KUKA KRL program: MyProgram_284().src

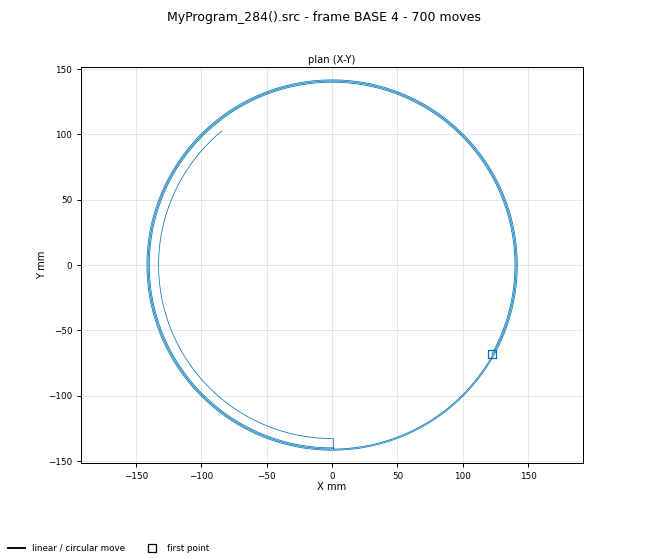
[picture p0: tool path of MyProgram_284().src in frame BASE 4, 700 of 700 moves have a stored position in this frame; points joined in program order, loops and branches not executed]
&ACCESS RVP
&REL 1
&PARAM TEMPLATE = C:\KRC\Roboter\Template\vorgabe
&PARAM EDITMASK = *
DEF MyProgram_284()
; ---- Setting reference (Base) ----
$BASE = BASE_DATA[4]

; --------------------------
; ---- Setting tool (TCP) ----
$TOOL = TOOL_DATA[3]
; --------------------------

$VEL.CP = VEL_APROX_PRINT
Startdeposition()
$VEL.CP = VEL_PRINT
LIN {X 122.1993,Y -68.1495,Z 174,A -26.2551,B 7.7078,C 0.3215,E1 7.8551,E2 478.0769} C_DIS
LIN {X 124.5651,Y -63.7171,Z 174,A -24.1572,B 7.7081,C 0.3154,E1 7.8578,E2 475.9716} C_DIS
LIN {X 126.1549,Y -60.5084,Z 174,A -22.4865,B 7.7084,C 0.3073,E1 7.8599,E2 474.2724} C_DIS
LIN {X 127.9066,Y -56.7133,Z 174,A -21.1789,B 7.7083,C 0.311,E1 7.8613,E2 473.0165} C_DIS
LIN {X 129.634,Y -52.6447,Z 174,A -19.4311,B 7.7083,C 0.3074,E1 7.8632,E2 471.2751} C_DIS
LIN {X 131.5394,Y -47.684,Z 174,A -17.3231,B 7.7086,C 0.3029,E1 7.8652,E2 469.1739} C_DIS
LIN {X 132.6761,Y -44.4231,Z 174,A -15.9508,B 7.7086,C 0.2999,E1 7.8665,E2 467.8057} C_DIS
LIN {X 133.516,Y -41.8378,Z 174,A -14.7782,B 7.7089,C 0.2956,E1 7.8675,E2 466.6243} C_DIS
LIN {X 135.2272,Y -35.9162,Z 174,A -12.5229,B 7.7089,C 0.294,E1 7.8692,E2 464.4017} C_DIS
LIN {X 136.3459,Y -31.4041,Z 174,A -10.4646,B 7.7092,C 0.2855,E1 7.8705,E2 462.3215} C_DIS
LIN {X 137.1536,Y -27.6644,Z 174,A -8.7503,B 7.7095,C 0.278,E1 7.8715,E2 460.5863} C_DIS
LIN {X 138.1088,Y -22.4214,Z 174,A -6.7596,B 7.7095,C 0.2757,E1 7.8725,E2 458.6188} C_DIS
LIN {X 138.6815,Y -18.5466,Z 174,A -5.2004,B 7.7097,C 0.2721,E1 7.8731,E2 457.0639} C_DIS
LIN {X 139.1996,Y -14.1607,Z 174,A -3.1875,B 7.71,C 0.2626,E1 7.8737,E2 455.0226} C_DIS
LIN {X 139.4882,Y -10.9545,Z 174,A -1.9592,B 7.7101,C 0.2607,E1 7.8739,E2 453.8049} C_DIS
LIN {X 139.7863,Y -6.0486,Z 174,A -0.0924,B 7.7102,C 0.2579,E1 7.8742,E2 451.9554} C_DIS
LIN {X 139.9098,Y -1.4915,Z 174,A 1.6918,B 7.7103,C 0.2542,E1 7.8742,E2 450.1803} C_DIS
LIN {X 139.8656,Y 3.7505,Z 174,A 3.9953,B 7.7106,C 0.2448,E1 7.8742,E2 447.8544} C_DIS
LIN {X 139.6455,Y 8.6938,Z 174,A 5.8419,B 7.7106,C 0.2427,E1 7.8739,E2 446.0296} C_DIS
LIN {X 139.3207,Y 12.8988,Z 174,A 7.2965,B 7.7106,C 0.2433,E1 7.8736,E2 444.6089} C_DIS
LIN {X 138.8413,Y 17.3162,Z 174,A 9.4268,B 7.711,C 0.2317,E1 7.8729,E2 442.4369} C_DIS
LIN {X 137.6741,Y 24.9464,Z 174,A 12.3433,B 7.7111,C 0.2278,E1 7.8716,E2 439.5497} C_DIS
LIN {X 136.0253,Y 32.7637,Z 174,A 15.5132,B 7.7113,C 0.2207,E1 7.8697,E2 436.3907} C_DIS
LIN {X 135.2183,Y 35.9496,Z 174,A 16.8457,B 7.7114,C 0.2172,E1 7.8688,E2 435.0589} C_DIS
LIN {X 134.3574,Y 39.045,Z 174,A 18.167,B 7.7116,C 0.2135,E1 7.8678,E2 433.7359} C_DIS
LIN {X 133.4759,Y 41.9634,Z 174,A 19.4631,B 7.7116,C 0.2091,E1 7.8667,E2 432.4328} C_DIS
LIN {X 132.2647,Y 45.6334,Z 174,A 20.9077,B 7.7117,C 0.2076,E1 7.8654,E2 431.0049} C_DIS
LIN {X 131.2197,Y 48.5594,Z 174,A 22.2206,B 7.7118,C 0.2033,E1 7.8641,E2 429.686} C_DIS
LIN {X 129.941,Y 51.8831,Z 174,A 24.4494,B 7.7123,C 0.1838,E1 7.8617,E2 427.3561} C_DIS
LIN {X 127.4014,Y 57.8428,Z 174,A 26.6346,B 7.7123,C 0.1864,E1 7.8593,E2 425.2304} C_DIS
LIN {X 125.7153,Y 61.4186,Z 174,A 27.8606,B 7.7122,C 0.1901,E1 7.8579,E2 424.0542} C_DIS
LIN {X 124.1071,Y 64.6062,Z 174,A 29.3051,B 7.7122,C 0.1868,E1 7.856,E2 422.6111} C_DIS
LIN {X 122.3418,Y 67.8921,Z 174,A 31.3586,B 7.7126,C 0.1724,E1 7.8531,E2 420.4888} C_DIS
LIN {X 119.7806,Y 72.315,Z 174,A 32.9061,B 7.7124,C 0.1782,E1 7.851,E2 419.0109} C_DIS
LIN {X 117.2705,Y 76.3185,Z 174,A 34.6702,B 7.7124,C 0.1769,E1 7.8484,E2 417.2678} C_DIS
LIN {X 115.0409,Y 79.6401,Z 174,A 36.4617,B 7.7126,C 0.17,E1 7.8456,E2 415.4559} C_DIS
LIN {X 112.3183,Y 83.4354,Z 174,A 38.1328,B 7.7126,C 0.1703,E1 7.8429,E2 413.8149} C_DIS
LIN {X 110.0921,Y 86.3509,Z 174,A 40.1246,B 7.7129,C 0.1573,E1 7.8393,E2 411.7595} C_DIS
LIN {X 107.4607,Y 89.6059,Z 174,A 41.515,B 7.7129,C 0.1599,E1 7.8369,E2 410.4102} C_DIS
LIN {X 104.7041,Y 92.8113,Z 174,A 43.4594,B 7.713,C 0.152,E1 7.8333,E2 408.4378} C_DIS
LIN {X 102.1452,Y 95.6208,Z 174,A 44.6972,B 7.713,C 0.1549,E1 7.831,E2 407.2404} C_DIS
LIN {X 99.0411,Y 98.8322,Z 174,A 46.4208,B 7.713,C 0.1532,E1 7.8277,E2 405.5298} C_DIS
LIN {X 94.8635,Y 102.8485,Z 174,A 48.8946,B 7.7131,C 0.1466,E1 7.8226,E2 403.0426} C_DIS
LIN {X 91.3702,Y 105.9639,Z 174,A 50.7297,B 7.7131,C 0.1446,E1 7.8188,E2 401.2174} C_DIS
LIN {X 88.0563,Y 108.7337,Z 174,A 52.5226,B 7.7132,C 0.1409,E1 7.8149,E2 399.421} C_DIS
LIN {X 84.604,Y 111.4413,Z 174,A 54.3131,B 7.7132,C 0.1379,E1 7.8109,E2 397.6311} C_DIS
LIN {X 80.4569,Y 114.4709,Z 174,A 56.6668,B 7.7134,C 0.1296,E1 7.8055,E2 395.2449} C_DIS
LIN {X 77.2065,Y 116.6881,Z 174,A 57.992,B 7.7134,C 0.1325,E1 7.8025,E2 393.9562} C_DIS
LIN {X 73.4825,Y 119.0685,Z 174,A 59.8229,B 7.7134,C 0.1293,E1 7.7982,E2 392.1225} C_DIS
LIN {X 69.1583,Y 121.6306,Z 174,A 61.7597,B 7.7134,C 0.1286,E1 7.7935,E2 390.2011} C_DIS
LIN {X 66.0546,Y 123.3437,Z 174,A 63.2273,B 7.7134,C 0.1264,E1 7.7899,E2 388.7314} C_DIS
LIN {X 58.451,Y 127.1215,Z 174,A 66.6086,B 7.7135,C 0.1238,E1 7.7815,E2 385.3624} C_DIS
LIN {X 52.7496,Y 129.5917,Z 174,A 69.091,B 7.7135,C 0.1221,E1 7.7751,E2 382.8883} C_DIS
LIN {X 49.4162,Y 130.8987,Z 174,A 70.6147,B 7.7135,C 0.1195,E1 7.7711,E2 381.3573} C_DIS
LIN {X 46.0839,Y 132.1085,Z 174,A 71.9894,B 7.7135,C 0.1195,E1 7.7675,E2 379.9926} C_DIS
LIN {X 43.2163,Y 133.0757,Z 174,A 73.315,B 7.7136,C 0.1169,E1 7.764,E2 378.6564} C_DIS
LIN {X 39.8202,Y 134.1304,Z 174,A 74.7349,B 7.7136,C 0.1163,E1 7.7602,E2 377.2413} C_DIS
LIN {X 36.1319,Y 135.1697,Z 174,A 76.2357,B 7.7136,C 0.1163,E1 7.7562,E2 375.7495} C_DIS
LIN {X 32.151,Y 136.1728,Z 174,A 78.6804,B 7.7138,C 0.1016,E1 7.7493,E2 373.2079} C_DIS
LIN {X 26.4354,Y 137.3957,Z 174,A 80.31,B 7.7137,C 0.1138,E1 7.7451,E2 371.6764} C_DIS
LIN {X 19.3821,Y 138.5673,Z 174,A 83.3147,B 7.7137,C 0.1112,E1 7.7368,E2 368.663} C_DIS
LIN {X 13.9273,Y 139.222,Z 174,A 85.559,B 7.7137,C 0.1106,E1 7.7306,E2 366.4202} C_DIS
LIN {X 10.1279,Y 139.5487,Z 174,A 87.0357,B 7.7137,C 0.1117,E1 7.7265,E2 364.9547} C_DIS
LIN {X 5.4892,Y 139.8081,Z 174,A 89.1817,B 7.7137,C 0.1073,E1 7.7204,E2 362.7787} C_DIS
LIN {X 0.3109,Y 139.9163,Z 174,A 91.1091,B 7.7137,C 0.1105,E1 7.7151,E2 360.8768} C_DIS
LIN {X -3.9902,Y 139.859,Z 174,A 92.7867,B 7.7137,C 0.112,E1 7.7104,E2 359.2106} C_DIS
LIN {X -9.1606,Y 139.6167,Z 174,A 94.922,B 7.7137,C 0.1121,E1 7.7045,E2 357.0744} C_DIS
LIN {X -14.8422,Y 139.1263,Z 174,A 97.3717,B 7.7137,C 0.1108,E1 7.6976,E2 354.6115} C_DIS
LIN {X -19.4903,Y 138.5519,Z 174,A 99.8517,B 7.7138,C 0.1022,E1 7.6906,E2 352.0612} C_DIS
LIN {X -24.6926,Y 137.7195,Z 174,A 101.2095,B 7.7136,C 0.1165,E1 7.6871,E2 350.8061} C_DIS
LIN {X -27.3108,Y 137.2255,Z 174,A 102.6319,B 7.7136,C 0.1117,E1 7.6831,E2 349.3427} C_DIS
LIN {X -32.0121,Y 136.2065,Z 174,A 104.56,B 7.7136,C 0.1136,E1 7.6779,E2 347.4211} C_DIS
LIN {X -35.8048,Y 135.2569,Z 174,A 106.0409,B 7.7136,C 0.1167,E1 7.6739,E2 345.9564} C_DIS
LIN {X -39.1445,Y 134.3282,Z 174,A 107.4312,B 7.7136,C 0.1183,E1 7.6702,E2 344.5707} C_DIS
LIN {X -42.3981,Y 133.337,Z 174,A 108.8728,B 7.7136,C 0.1187,E1 7.6663,E2 343.1239} C_DIS
LIN {X -45.0988,Y 132.4501,Z 174,A 110.163,B 7.7136,C 0.1178,E1 7.6629,E2 341.8187} C_DIS
LIN {X -50.4383,Y 130.5081,Z 174,A 113.0061,B 7.7136,C 0.1119,E1 7.6553,E2 338.9116} C_DIS
LIN {X -55.163,Y 128.5827,Z 174,A 114.3244,B 7.7135,C 0.1265,E1 7.6522,E2 337.6926} C_DIS
LIN {X -61.6152,Y 125.6183,Z 174,A 117.4422,B 7.7135,C 0.1268,E1 7.6442,E2 334.5507} C_DIS
LIN {X -64.8167,Y 123.9965,Z 174,A 118.9194,B 7.7135,C 0.1286,E1 7.6405,E2 333.0738} C_DIS
LIN {X -67.5389,Y 122.5374,Z 174,A 120.7434,B 7.7135,C 0.1217,E1 7.6359,E2 331.18} C_DIS
LIN {X -71.6524,Y 120.1781,Z 174,A 122.2439,B 7.7134,C 0.1314,E1 7.6324,E2 329.7372} C_DIS
LIN {X -74.8429,Y 118.2177,Z 174,A 123.8797,B 7.7134,C 0.1322,E1 7.6285,E2 328.0898} C_DIS
LIN {X -79.0031,Y 115.479,Z 174,A 125.8589,B 7.7133,C 0.1364,E1 7.624,E2 326.12} C_DIS
LIN {X -81.9231,Y 113.4262,Z 174,A 127.1872,B 7.7133,C 0.1409,E1 7.621,E2 324.8098} C_DIS
LIN {X -85.236,Y 110.9577,Z 174,A 129.4591,B 7.7133,C 0.1351,E1 7.6158,E2 322.4658} C_DIS
LIN {X -88.7884,Y 108.1368,Z 174,A 130.9257,B 7.7131,C 0.1444,E1 7.6127,E2 321.0506} C_DIS
LIN {X -94.8734,Y 102.8394,Z 174,A 134.9758,B 7.7132,C 0.1396,E1 7.6041,E2 316.9084} C_DIS
LIN {X -99.2376,Y 98.6344,Z 174,A 136.7497,B 7.7129,C 0.1553,E1 7.6008,E2 315.2271} C_DIS
LIN {X -104.5185,Y 93.021,Z 174,A 140.4374,B 7.7129,C 0.1541,E1 7.5937,E2 311.4749} C_DIS
LIN {X -107.56,Y 89.4863,Z 174,A 141.9414,B 7.7127,C 0.1644,E1 7.5911,E2 310.0243} C_DIS
LIN {X -110.7442,Y 85.5136,Z 174,A 144.0936,B 7.7127,C 0.1681,E1 7.5874,E2 307.8657} C_DIS
LIN {X -113.4608,Y 81.8753,Z 174,A 145.8871,B 7.7126,C 0.1734,E1 7.5844,E2 306.0823} C_DIS
LIN {X -115.9587,Y 78.2972,Z 174,A 147.7171,B 7.7125,C 0.1771,E1 7.5815,E2 304.2486} C_DIS
LIN {X -119.4121,Y 72.9224,Z 174,A 150.4658,B 7.7124,C 0.1816,E1 7.5774,E2 301.4856} C_DIS
LIN {X -121.5604,Y 69.2814,Z 174,A 152.2284,B 7.7123,C 0.1855,E1 7.5749,E2 299.7208} C_DIS
LIN {X -123.7428,Y 65.2999,Z 174,A 153.9528,B 7.7121,C 0.1921,E1 7.5727,E2 298.0153} C_DIS
LIN {X -125.3067,Y 62.2467,Z 174,A 155.2919,B 7.712,C 0.1967,E1 7.571,E2 296.6858} C_DIS
LIN {X -127.1646,Y 58.3576,Z 174,A 157.2294,B 7.712,C 0.1989,E1 7.5687,E2 294.7282} C_DIS
LIN {X -128.8679,Y 54.4954,Z 174,A 159.0105,B 7.7118,C 0.2027,E1 7.5667,E2 292.9421} C_DIS
LIN {X -130.2987,Y 50.9768,Z 174,A 160.5654,B 7.7118,C 0.2069,E1 7.5651,E2 291.3888} C_DIS
LIN {X -131.5535,Y 47.645,Z 174,A 161.9957,B 7.7116,C 0.2113,E1 7.5637,E2 289.9634} C_DIS
LIN {X -132.5578,Y 44.7784,Z 174,A 163.4094,B 7.7116,C 0.2123,E1 7.5624,E2 288.5293} C_DIS
LIN {X -133.7726,Y 41.0028,Z 174,A 164.8584,B 7.7114,C 0.2192,E1 7.5612,E2 287.1042} C_DIS
LIN {X -134.5659,Y 38.325,Z 174,A 166.2505,B 7.7114,C 0.2189,E1 7.5601,E2 285.6815} C_DIS
LIN {X -135.5606,Y 34.6371,Z 174,A 167.6747,B 7.7112,C 0.2253,E1 7.5591,E2 284.2767} C_DIS
LIN {X -136.3128,Y 31.5488,Z 174,A 169.0655,B 7.7112,C 0.2277,E1 7.5582,E2 282.8757} C_DIS
LIN {X -137.1859,Y 27.5054,Z 174,A 170.9807,B 7.7111,C 0.2294,E1 7.5571,E2 280.9338} C_DIS
LIN {X -137.9905,Y 23.1304,Z 174,A 172.9016,B 7.711,C 0.2331,E1 7.5562,E2 279.0018} C_DIS
LIN {X -138.5009,Y 19.8468,Z 174,A 174.0154,B 7.7108,C 0.2405,E1 7.5558,E2 277.921} C_DIS
LIN {X -138.92,Y 16.663,Z 174,A 176.0497,B 7.711,C 0.2341,E1 7.5551,E2 275.7953} C_DIS
LIN {X -139.485,Y 10.9969,Z 174,A 177.6762,B 7.7104,C 0.2508,E1 7.5547,E2 274.262} C_DIS
LIN {X -139.8535,Y 4.1888,Z 174,A -179.5152,B 7.7102,C 0.2586,E1 7.5544,E2 271.4538} C_DIS
LIN {X -139.8767,Y -3.3537,Z 174,A -176.4156,B 7.7099,C 0.2674,E1 7.5544,E2 268.3557} C_DIS
LIN {X -139.6037,Y -9.3711,Z 174,A -173.803,B 7.7097,C 0.2725,E1 7.5547,E2 265.7267} C_DIS
LIN {X -139.2586,Y -13.5457,Z 174,A -171.5038,B 7.7098,C 0.2691,E1 7.5554,E2 263.3534} C_DIS
LIN {X -138.7428,Y -18.0786,Z 174,A -170.1635,B 7.7094,C 0.2819,E1 7.5558,E2 262.0829} C_DIS
LIN {X -138.2464,Y -21.5488,Z 174,A -168.6175,B 7.7093,C 0.2844,E1 7.5564,E2 260.5238} C_DIS
LIN {X -137.4895,Y -25.9446,Z 174,A -166.7279,B 7.7091,C 0.2887,E1 7.5574,E2 258.6275} C_DIS
LIN {X -136.7177,Y -29.7437,Z 174,A -165.1322,B 7.709,C 0.293,E1 7.5583,E2 257.0319} C_DIS
LIN {X -135.672,Y -34.1983,Z 174,A -163.2641,B 7.7088,C 0.2983,E1 7.5595,E2 255.166} C_DIS
LIN {X -134.7995,Y -37.4896,Z 174,A -161.8425,B 7.7086,C 0.3018,E1 7.5606,E2 253.7419} C_DIS
LIN {X -133.7455,Y -41.0912,Z 174,A -160.2955,B 7.7085,C 0.3058,E1 7.5618,E2 252.1946} C_DIS
LIN {X -132.8248,Y -43.9766,Z 174,A -159.0212,B 7.7083,C 0.3087,E1 7.5629,E2 250.9168} C_DIS
LIN {X -130.9912,Y -49.1695,Z 174,A -156.7748,B 7.7081,C 0.3149,E1 7.565,E2 248.673} C_DIS
LIN {X -129.1941,Y -53.7144,Z 174,A -154.6747,B 7.7079,C 0.3187,E1 7.5672,E2 246.5614} C_DIS
LIN {X -127.8613,Y -56.8145,Z 174,A -153.3105,B 7.7078,C 0.3226,E1 7.5688,E2 245.2005} C_DIS
LIN {X -126.4013,Y -59.9927,Z 174,A -151.8707,B 7.7076,C 0.3262,E1 7.5705,E2 243.7605} C_DIS
LIN {X -124.9,Y -63.0594,Z 174,A -150.3827,B 7.7076,C 0.3284,E1 7.5723,E2 242.2617} C_DIS
LIN {X -121.4694,Y -69.441,Z 174,A -147.0513,B 7.7075,C 0.3304,E1 7.5769,E2 238.8845} C_DIS
LIN {X -119.6565,Y -72.5202,Z 174,A -145.8253,B 7.7071,C 0.3375,E1 7.5786,E2 237.6903} C_DIS
LIN {X -117.7583,Y -75.5636,Z 174,A -144.2927,B 7.7071,C 0.34,E1 7.5809,E2 236.15} C_DIS
LIN {X -115.1881,Y -79.4269,Z 174,A -142.3909,B 7.7068,C 0.3444,E1 7.5839,E2 234.2489} C_DIS
LIN {X -112.6633,Y -82.969,Z 174,A -140.5791,B 7.7067,C 0.348,E1 7.5869,E2 232.4339} C_DIS
LIN {X -109.8304,Y -86.6847,Z 174,A -138.6388,B 7.7065,C 0.3519,E1 7.5902,E2 230.4909} C_DIS
LIN {X -106.9266,Y -90.2425,Z 174,A -136.826,B 7.7063,C 0.3569,E1 7.5934,E2 228.6876} C_DIS
LIN {X -100.9439,Y -96.8878,Z 174,A -133.3214,B 7.7058,C 0.3669,E1 7.6,E2 225.205} C_DIS
LIN {X -96.8585,Y -100.972,Z 174,A -130.5985,B 7.7058,C 0.3661,E1 7.6055,E2 222.4362} C_DIS
LIN {X -93.4578,Y -104.1274,Z 174,A -128.6954,B 7.7057,C 0.3695,E1 7.6094,E2 220.5332} C_DIS
LIN {X -90.2245,Y -106.9417,Z 174,A -126.8866,B 7.7056,C 0.3719,E1 7.6132,E2 218.7177} C_DIS
LIN {X -86.6677,Y -109.8437,Z 174,A -124.993,B 7.7054,C 0.3749,E1 7.6173,E2 216.8226} C_DIS
LIN {X -83.1559,Y -112.526,Z 174,A -122.6402,B 7.7057,C 0.3692,E1 7.6228,E2 214.3985} C_DIS
LIN {X -78.8921,Y -115.5551,Z 174,A -121.022,B 7.7051,C 0.3809,E1 7.6263,E2 212.8497} C_DIS
LIN {X -76.4311,Y -117.1973,Z 174,A -119.6907,B 7.7051,C 0.3808,E1 7.6295,E2 211.5028} C_DIS
LIN {X -72.0195,Y -119.9593,Z 174,A -117.6103,B 7.705,C 0.3846,E1 7.6344,E2 209.4292} C_DIS
LIN {X -68.5029,Y -122.0009,Z 174,A -114.5497,B 7.706,C 0.3639,E1 7.6424,E2 206.1828} C_DIS
LIN {X -59.5873,Y -126.595,Z 174,A -111.4654,B 7.7049,C 0.3856,E1 7.6498,E2 203.2354} C_DIS
LIN {X -55.8459,Y -128.2874,Z 174,A -110.2438,B 7.7044,C 0.395,E1 7.6528,E2 202.0744} C_DIS
LIN {X -52.628,Y -129.6407,Z 174,A -108.7445,B 7.7044,C 0.3953,E1 7.6566,E2 200.5658} C_DIS
LIN {X -49.2852,Y -130.9478,Z 174,A -107.4134,B 7.7042,C 0.3989,E1 7.6601,E2 199.2528} C_DIS
LIN {X -46.4697,Y -131.9748,Z 174,A -105.9801,B 7.7044,C 0.3965,E1 7.6639,E2 197.7922} C_DIS
LIN {X -42.785,Y -133.2134,Z 174,A -104.4603,B 7.7042,C 0.399,E1 7.6679,E2 196.2816} C_DIS
LIN {X -39.4044,Y -134.2521,Z 174,A -103.0782,B 7.7042,C 0.4011,E1 7.6716,E2 194.9079} C_DIS
LIN {X -35.1154,Y -135.4386,Z 174,A -100.8009,B 7.7045,C 0.3946,E1 7.6779,E2 192.5701} C_DIS
LIN {X -31.4193,Y -136.3424,Z 174,A -99.5706,B 7.7041,C 0.401,E1 7.6811,E2 191.3828} C_DIS
LIN {X -27.3221,Y -137.2232,Z 174,A -97.9868,B 7.704,C 0.4041,E1 7.6854,E2 189.816} C_DIS
LIN {X -22.2894,Y -138.1308,Z 174,A -95.7605,B 7.704,C 0.4026,E1 7.6916,E2 187.5717} C_DIS
LIN {X -18.372,Y -138.7044,Z 174,A -94.1906,B 7.704,C 0.4039,E1 7.6959,E2 186.0079} C_DIS
LIN {X -15.1561,Y -139.0925,Z 174,A -92.8136,B 7.704,C 0.4033,E1 7.6998,E2 184.6238} C_DIS
LIN {X -11.1877,Y -139.469,Z 174,A -91.1227,B 7.704,C 0.4025,E1 7.7045,E2 182.9246} C_DIS
LIN {X -7.2495,Y -139.7281,Z 174,A -89.5868,B 7.704,C 0.404,E1 7.7087,E2 181.3985} C_DIS
LIN {X -3.6909,Y -139.8673,Z 174,A -88.126,B 7.704,C 0.404,E1 7.7128,E2 179.9368} C_DIS
LIN {X 0.9946,Y -139.9107,Z 174,A -86.3405,B 7.7039,C 0.4061,E1 7.7178,E2 178.1679} C_DIS
Enddeposition()
LIN {X 0.9946,Y -139.9107,Z 174,A -86.3405,B 7.7039,C 0.4061,E1 7.7178,E2 178.1679} C_DIS
Startdeposition()
$VEL.CP = VEL_PRINT
LIN {X -0.9199,Y -140.8201,Z 174,A -87.6311,B 7.7029,C 0.4197,E1 7.7137,E2 179.56} C_DIS
LIN {X -5.2754,Y -140.7243,Z 174,A -89.3929,B 7.7029,C 0.4197,E1 7.7088,E2 181.3211} C_DIS
LIN {X -9.1302,Y -140.5274,Z 174,A -91.0599,B 7.7029,C 0.4212,E1 7.7041,E2 183.0016} C_DIS
LIN {X -13.3615,Y -140.1876,Z 174,A -92.7206,B 7.7029,C 0.4199,E1 7.6995,E2 184.6541} C_DIS
LIN {X -17.616,Y -139.7183,Z 174,A -94.3536,B 7.703,C 0.4176,E1 7.695,E2 186.2736} C_DIS
LIN {X -20.6042,Y -139.309,Z 174,A -95.7976,B 7.7029,C 0.421,E1 7.6909,E2 187.7466} C_DIS
LIN {X -25.5092,Y -138.4946,Z 174,A -97.6582,B 7.703,C 0.4175,E1 7.6858,E2 189.5864} C_DIS
LIN {X -28.593,Y -137.8903,Z 174,A -98.9253,B 7.703,C 0.4167,E1 7.6824,E2 190.8524} C_DIS
LIN {X -31.9929,Y -137.1419,Z 174,A -100.3442,B 7.7031,C 0.416,E1 7.6785,E2 192.272} C_DIS
LIN {X -35.4789,Y -136.2826,Z 174,A -102.1567,B 7.7029,C 0.4211,E1 7.6735,E2 194.131} C_DIS
LIN {X -38.7987,Y -135.3747,Z 174,A -103.2295,B 7.7032,C 0.4146,E1 7.6707,E2 195.1612} C_DIS
LIN {X -42.0658,Y -134.3954,Z 174,A -104.7828,B 7.7032,C 0.4164,E1 7.6665,E2 196.7365} C_DIS
LIN {X -46.2905,Y -132.997,Z 174,A -106.4863,B 7.7032,C 0.4131,E1 7.662,E2 198.4262} C_DIS
LIN {X -50.2719,Y -131.546,Z 174,A -108.1792,B 7.7034,C 0.4111,E1 7.6576,E2 200.1152} C_DIS
LIN {X -53.0089,Y -130.4652,Z 174,A -109.4897,B 7.7034,C 0.4118,E1 7.6542,E2 201.4407} C_DIS
LIN {X -57.0105,Y -128.7674,Z 174,A -111.3907,B 7.7034,C 0.4121,E1 7.6493,E2 203.3591} C_DIS
LIN {X -61.281,Y -126.7912,Z 174,A -113.198,B 7.7035,C 0.4082,E1 7.6447,E2 205.1526} C_DIS
LIN {X -65.1406,Y -124.851,Z 174,A -115.3883,B 7.7033,C 0.413,E1 7.6392,E2 207.3993} C_DIS
LIN {X -69.1803,Y -122.6607,Z 174,A -116.6186,B 7.7039,C 0.4003,E1 7.6364,E2 208.5461} C_DIS
LIN {X -71.8913,Y -121.0918,Z 174,A -118.1687,B 7.7039,C 0.403,E1 7.6325,E2 210.1324} C_DIS
LIN {X -75.7607,Y -118.7092,Z 174,A -120.0031,B 7.7039,C 0.4001,E1 7.6282,E2 211.9647} C_DIS
LIN {X -79.4472,Y -116.2744,Z 174,A -121.8516,B 7.7041,C 0.3982,E1 7.6239,E2 213.8197} C_DIS
LIN {X -83.4437,Y -113.4401,Z 174,A -123.6854,B 7.7043,C 0.3925,E1 7.6198,E2 215.6324} C_DIS
LIN {X -86.3954,Y -111.2087,Z 174,A -125.3768,B 7.7043,C 0.3929,E1 7.616,E2 217.3478} C_DIS
LIN {X -90.0889,Y -108.2388,Z 174,A -127.3058,B 7.7045,C 0.3896,E1 7.6118,E2 219.2765} C_DIS
LIN {X -93.1826,Y -105.5866,Z 174,A -129.0055,B 7.7046,C 0.3872,E1 7.6082,E2 220.9813} C_DIS
LIN {X -96.5887,Y -102.4799,Z 174,A -130.9856,B 7.7047,C 0.3853,E1 7.6041,E2 222.9745} C_DIS
LIN {X -100.0974,Y -99.056,Z 174,A -132.9204,B 7.7049,C 0.3805,E1 7.6003,E2 224.9009} C_DIS
LIN {X -103.2747,Y -95.7389,Z 174,A -134.7848,B 7.7051,C 0.3766,E1 7.5967,E2 226.7642} C_DIS
LIN {X -106.87,Y -91.7081,Z 174,A -136.7369,B 7.7055,C 0.3683,E1 7.5932,E2 228.6836} C_DIS
LIN {X -110.0201,Y -87.9043,Z 174,A -139.1084,B 7.7055,C 0.3694,E1 7.5889,E2 231.1014} C_DIS
LIN {X -112.87,Y -84.2134,Z 174,A -141.0002,B 7.7057,C 0.3651,E1 7.5857,E2 232.9917} C_DIS
LIN {X -115.4727,Y -80.6078,Z 174,A -142.8449,B 7.7059,C 0.3615,E1 7.5827,E2 234.8402} C_DIS
LIN {X -117.9834,Y -76.8862,Z 174,A -144.7834,B 7.7059,C 0.3589,E1 7.5797,E2 236.7924} C_DIS
LIN {X -120.2021,Y -73.3694,Z 174,A -146.4053,B 7.7062,C 0.3538,E1 7.5774,E2 238.4044} C_DIS
LIN {X -124.6963,Y -65.4352,Z 174,A -149.7659,B 7.7069,C 0.3395,E1 7.5728,E2 241.7176} C_DIS
LIN {X -126.4043,Y -62.0722,Z 174,A -151.6773,B 7.7068,C 0.3411,E1 7.5704,E2 243.6771} C_DIS
LIN {X -128.0913,Y -58.5148,Z 174,A -153.2747,B 7.707,C 0.3369,E1 7.5685,E2 245.273} C_DIS
LIN {X -129.5364,Y -55.2429,Z 174,A -154.7715,B 7.7071,C 0.3337,E1 7.5668,E2 246.7743} C_DIS
LIN {X -130.9597,Y -51.78,Z 174,A -156.2974,B 7.7073,C 0.3298,E1 7.5652,E2 248.2996} C_DIS
LIN {X -132.1568,Y -48.6434,Z 174,A -157.8289,B 7.7073,C 0.3285,E1 7.5637,E2 249.8516} C_DIS
LIN {X -133.1982,Y -45.7102,Z 174,A -158.9966,B 7.7075,C 0.3237,E1 7.5626,E2 251.0056} C_DIS
LIN {X -134.2115,Y -42.6417,Z 174,A -160.3914,B 7.7076,C 0.3212,E1 7.5614,E2 252.4098} C_DIS
LIN {X -135.3455,Y -38.8984,Z 174,A -161.9565,B 7.7078,C 0.3165,E1 7.5602,E2 253.9704} C_DIS
LIN {X -136.148,Y -35.9837,Z 174,A -163.2525,B 7.7079,C 0.314,E1 7.5592,E2 255.274} C_DIS
LIN {X -137.3089,Y -31.2618,Z 174,A -165.2148,B 7.7082,C 0.3083,E1 7.558,E2 257.2328} C_DIS
LIN {X -138.0564,Y -27.777,Z 174,A -166.7003,B 7.7082,C 0.3047,E1 7.5571,E2 258.7216} C_DIS
LIN {X -138.7388,Y -24.1461,Z 174,A -168.3906,B 7.7084,C 0.3032,E1 7.5563,E2 260.4349} C_DIS
LIN {X -139.4753,Y -19.4403,Z 174,A -170.8208,B 7.7084,C 0.3045,E1 7.5553,E2 262.9263} C_DIS
LIN {X -140.0872,Y -14.3914,Z 174,A -172.2697,B 7.7089,C 0.29,E1 7.5549,E2 264.2944} C_DIS
LIN {X -140.343,Y -11.6186,Z 174,A -173.4381,B 7.7089,C 0.2872,E1 7.5546,E2 265.4664} C_DIS
LIN {X -140.5769,Y -8.3268,Z 174,A -174.8349,B 7.7091,C 0.2841,E1 7.5543,E2 266.869} C_DIS
LIN {X -140.7513,Y -4.534,Z 174,A -176.6274,B 7.7091,C 0.2831,E1 7.5541,E2 268.6918} C_DIS
LIN {X -140.8022,Y 2.4189,Z 174,A -179.326,B 7.7095,C 0.2732,E1 7.5541,E2 271.3713} C_DIS
LIN {X -140.6973,Y 5.9661,Z 174,A 179.2534,B 7.7096,C 0.2687,E1 7.5543,E2 272.7877} C_DIS
LIN {X -140.5038,Y 9.5045,Z 174,A 177.593,B 7.7096,C 0.2676,E1 7.5546,E2 274.4747} C_DIS
LIN {X -139.9436,Y 15.7175,Z 174,A 175.2161,B 7.71,C 0.258,E1 7.5552,E2 276.8287} C_DIS
LIN {X -139.6205,Y 18.3626,Z 174,A 173.4354,B 7.7098,C 0.2647,E1 7.5559,E2 278.6968} C_DIS
LIN {X -138.857,Y 23.4493,Z 174,A 171.9933,B 7.7103,C 0.2496,E1 7.5565,E2 280.0545} C_DIS
LIN {X -137.7157,Y 29.4195,Z 174,A 169.6149,B 7.7105,C 0.2413,E1 7.5578,E2 282.4185} C_DIS
LIN {X -137.1065,Y 32.1479,Z 174,A 168.2663,B 7.7105,C 0.2411,E1 7.5586,E2 283.7931} C_DIS
LIN {X -135.9793,Y 36.6164,Z 174,A 166.3642,B 7.7107,C 0.2362,E1 7.5599,E2 285.6968} C_DIS
LIN {X -135.0193,Y 40.0125,Z 174,A 164.8168,B 7.7107,C 0.2338,E1 7.5611,E2 287.257} C_DIS
LIN {X -133.94,Y 43.4915,Z 174,A 163.3819,B 7.7109,C 0.229,E1 7.5623,E2 288.6844} C_DIS
LIN {X -133.0249,Y 46.2101,Z 174,A 162.1708,B 7.7109,C 0.2264,E1 7.5634,E2 289.8999} C_DIS
LIN {X -131.8122,Y 49.5637,Z 174,A 160.6429,B 7.7111,C 0.2236,E1 7.5649,E2 291.4362} C_DIS
LIN {X -130.5091,Y 52.9001,Z 174,A 159.2041,B 7.7111,C 0.2194,E1 7.5664,E2 292.8712} C_DIS
LIN {X -129.1196,Y 56.2069,Z 174,A 157.6486,B 7.7113,C 0.2169,E1 7.5681,E2 294.4376} C_DIS
LIN {X -127.346,Y 60.1196,Z 174,A 155.8845,B 7.7113,C 0.2125,E1 7.5702,E2 296.202} C_DIS
LIN {X -126.1171,Y 62.6544,Z 174,A 154.7625,B 7.7115,C 0.2092,E1 7.5716,E2 297.3197} C_DIS
LIN {X -124.0893,Y 66.5836,Z 174,A 152.8714,B 7.7115,C 0.2059,E1 7.5741,E2 299.2208} C_DIS
LIN {X -121.5874,Y 71.0502,Z 174,A 150.7047,B 7.7117,C 0.2018,E1 7.5771,E2 301.3961} C_DIS
LIN {X -118.105,Y 76.6989,Z 174,A 148.0906,B 7.7119,C 0.194,E1 7.5809,E2 303.9967} C_DIS
LIN {X -115.8103,Y 80.1226,Z 174,A 146.3157,B 7.7119,C 0.1914,E1 7.5837,E2 305.7823} C_DIS
LIN {X -113.4121,Y 83.4818,Z 174,A 144.6323,B 7.712,C 0.1875,E1 7.5865,E2 307.4647} C_DIS
LIN {X -110.5367,Y 87.254,Z 174,A 142.6991,B 7.7121,C 0.1831,E1 7.5898,E2 309.3964} C_DIS
LIN {X -105.8155,Y 92.9227,Z 174,A 139.8624,B 7.7123,C 0.174,E1 7.5948,E2 312.2095} C_DIS
LIN {X -100.9185,Y 98.2196,Z 174,A 136.9404,B 7.7125,C 0.1676,E1 7.6004,E2 315.1273} C_DIS
LIN {X -97.6136,Y 101.5051,Z 174,A 134.671,B 7.7125,C 0.1693,E1 7.605,E2 317.4421} C_DIS
LIN {X -94.5974,Y 104.3209,Z 174,A 132.6356,B 7.7124,C 0.1713,E1 7.6093,E2 319.5206} C_DIS
LIN {X -91.4787,Y 107.0664,Z 174,A 131.3771,B 7.7126,C 0.1617,E1 7.6118,E2 320.7235} C_DIS
LIN {X -85.197,Y 112.13,Z 174,A 127.5585,B 7.7126,C 0.1638,E1 7.6203,E2 324.6062} C_DIS
LIN {X -81.6889,Y 114.7106,Z 174,A 126.2421,B 7.7128,C 0.1539,E1 7.6232,E2 325.8642} C_DIS
LIN {X -78.3772,Y 116.9982,Z 174,A 124.4694,B 7.7128,C 0.1533,E1 7.6273,E2 327.6524} C_DIS
LIN {X -74.3547,Y 119.5947,Z 174,A 122.5308,B 7.7128,C 0.1501,E1 7.6319,E2 329.5881} C_DIS
LIN {X -70.3644,Y 121.9853,Z 174,A 120.5403,B 7.7128,C 0.1489,E1 7.6367,E2 331.5894} C_DIS
LIN {X -67.0663,Y 123.8297,Z 174,A 119.0371,B 7.7129,C 0.1462,E1 7.6404,E2 333.087} C_DIS
LIN {X -63.4288,Y 125.7298,Z 174,A 117.4604,B 7.7129,C 0.1425,E1 7.6442,E2 334.6507} C_DIS
LIN {X -58.4531,Y 128.1199,Z 174,A 115.2275,B 7.713,C 0.1396,E1 7.6499,E2 336.8803} C_DIS
LIN {X -55.4708,Y 129.4378,Z 174,A 113.8476,B 7.713,C 0.1389,E1 7.6534,E2 338.2659} C_DIS
LIN {X -51.7299,Y 130.9792,Z 174,A 112.2575,B 7.713,C 0.1362,E1 7.6575,E2 339.8477} C_DIS
LIN {X -45.4174,Y 133.2997,Z 174,A 109.4785,B 7.7131,C 0.1342,E1 7.6648,E2 342.6302} C_DIS
LIN {X -42.415,Y 134.2839,Z 174,A 108.0928,B 7.7131,C 0.1346,E1 7.6685,E2 344.0275} C_DIS
LIN {X -38.7309,Y 135.3943,Z 174,A 106.5043,B 7.7131,C 0.1337,E1 7.6728,E2 345.618} C_DIS
LIN {X -33.3248,Y 136.8232,Z 174,A 104.5035,B 7.7132,C 0.1276,E1 7.6781,E2 347.5827} C_DIS
LIN {X -26.2207,Y 138.3603,Z 174,A 100.9921,B 7.7132,C 0.1349,E1 7.6879,E2 351.1618} C_DIS
LIN {X -22.5118,Y 139.0134,Z 174,A 99.5705,B 7.7132,C 0.1324,E1 7.6918,E2 352.5688} C_DIS
LIN {X -17.4146,Y 139.7439,Z 174,A 97.5603,B 7.7132,C 0.1302,E1 7.6973,E2 354.5672} C_DIS
LIN {X -12.8003,Y 140.2415,Z 174,A 95.712,B 7.7132,C 0.129,E1 7.7024,E2 356.4095} C_DIS
LIN {X -9.6063,Y 140.4964,Z 174,A 94.5405,B 7.7132,C 0.1265,E1 7.7056,E2 357.5638} C_DIS
LIN {X -6.0489,Y 140.6941,Z 174,A 92.9583,B 7.7132,C 0.1285,E1 7.7101,E2 359.1619} C_DIS
LIN {X -2.2552,Y 140.805,Z 174,A 91.5409,B 7.7132,C 0.1263,E1 7.714,E2 360.5626} C_DIS
LIN {X 1.5905,Y 140.8159,Z 174,A 89.9252,B 7.7132,C 0.1271,E1 7.7185,E2 362.184} C_DIS
LIN {X 4.431,Y 140.7542,Z 174,A 88.7567,B 7.7132,C 0.1274,E1 7.7218,E2 363.3536} C_DIS
LIN {X 8.2831,Y 140.5796,Z 174,A 87.1612,B 7.7132,C 0.1281,E1 7.7263,E2 364.9518} C_DIS
LIN {X 12.6975,Y 140.2513,Z 174,A 85.4611,B 7.7132,C 0.1268,E1 7.731,E2 366.6386} C_DIS
LIN {X 15.4499,Y 139.9733,Z 174,A 84.304,B 7.7132,C 0.1277,E1 7.7342,E2 367.7992} C_DIS
LIN {X 18.5042,Y 139.6019,Z 174,A 82.9959,B 7.7132,C 0.1291,E1 7.7378,E2 369.114} C_DIS
LIN {X 23.5302,Y 138.8434,Z 174,A 80.9986,B 7.7132,C 0.1288,E1 7.7433,E2 371.1017} C_DIS
LIN {X 27.2279,Y 138.1677,Z 174,A 79.4846,B 7.7132,C 0.1294,E1 7.7475,E2 372.6135} C_DIS
LIN {X 30.5238,Y 137.4773,Z 174,A 78.1147,B 7.7132,C 0.1302,E1 7.7512,E2 373.983} C_DIS
LIN {X 35.1705,Y 136.3611,Z 174,A 76.2032,B 7.7132,C 0.1309,E1 7.7564,E2 375.8899} C_DIS
LIN {X 38.094,Y 135.5724,Z 174,A 74.9398,B 7.7132,C 0.1324,E1 7.7598,E2 377.1569} C_DIS
LIN {X 41.5282,Y 134.5605,Z 174,A 73.4118,B 7.7132,C 0.1349,E1 7.7639,E2 378.6937} C_DIS
LIN {X 45.261,Y 133.3532,Z 174,A 71.9063,B 7.7132,C 0.1347,E1 7.7678,E2 380.1876} C_DIS
LIN {X 47.8874,Y 132.4303,Z 174,A 70.7925,B 7.7131,C 0.1354,E1 7.7708,E2 381.2987} C_DIS
LIN {X 51.2916,Y 131.1496,Z 174,A 69.2591,B 7.7131,C 0.1379,E1 7.7748,E2 382.8388} C_DIS
LIN {X 55.4458,Y 129.4487,Z 174,A 67.6335,B 7.7131,C 0.1363,E1 7.7789,E2 384.4388} C_DIS
LIN {X 59.3907,Y 127.6863,Z 174,A 65.7179,B 7.713,C 0.1412,E1 7.7838,E2 386.3742} C_DIS
LIN {X 63.1678,Y 125.8627,Z 174,A 63.6013,B 7.7128,C 0.151,E1 7.7893,E2 388.5425} C_DIS
LIN {X 66.9838,Y 123.8743,Z 174,A 62.2125,B 7.7128,C 0.1467,E1 7.7926,E2 389.8858} C_DIS
LIN {X 70.9942,Y 121.6202,Z 174,A 60.433,B 7.7128,C 0.1476,E1 7.7969,E2 391.6537} C_DIS
LIN {X 74.1439,Y 119.7259,Z 174,A 58.9509,B 7.7128,C 0.1496,E1 7.8004,E2 393.1342} C_DIS
LIN {X 77.3678,Y 117.6679,Z 174,A 57.4098,B 7.7128,C 0.1517,E1 7.804,E2 394.6736} C_DIS
LIN {X 81.171,Y 115.0773,Z 174,A 55.5096,B 7.7128,C 0.1553,E1 7.8084,E2 396.5775} C_DIS
LIN {X 84.5948,Y 112.5847,Z 174,A 53.7914,B 7.7127,C 0.1581,E1 7.8122,E2 398.2953} C_DIS
LIN {X 88.112,Y 109.8541,Z 174,A 51.988,B 7.7127,C 0.1612,E1 7.8162,E2 400.098} C_DIS
LIN {X 91.6331,Y 106.9346,Z 174,A 50.1338,B 7.7125,C 0.1645,E1 7.8201,E2 401.9518} C_DIS
LIN {X 98.2137,Y 100.9243,Z 174,A 46.5737,B 7.7125,C 0.1703,E1 7.8274,E2 405.5045} C_DIS
LIN {X 101.1755,Y 97.9542,Z 174,A 44.9607,B 7.7124,C 0.172,E1 7.8305,E2 407.1061} C_DIS
LIN {X 104.0787,Y 94.8643,Z 174,A 43.1634,B 7.7123,C 0.177,E1 7.834,E2 408.9132} C_DIS
LIN {X 106.5318,Y 92.1008,Z 174,A 41.69,B 7.7123,C 0.1797,E1 7.8367,E2 410.3833} C_DIS
LIN {X 112.2349,Y 85.0583,Z 174,A 38.2231,B 7.7121,C 0.1836,E1 7.8427,E2 413.8237} C_DIS
LIN {X 114.4579,Y 82.0422,Z 174,A 36.5755,B 7.712,C 0.1896,E1 7.8454,E2 415.4876} C_DIS
LIN {X 117.109,Y 78.2113,Z 174,A 34.7638,B 7.7119,C 0.1924,E1 7.8482,E2 417.2895} C_DIS
LIN {X 119.4059,Y 74.6582,Z 174,A 33.0832,B 7.7119,C 0.1958,E1 7.8507,E2 418.9658} C_DIS
LIN {X 121.5442,Y 71.1237,Z 174,A 31.2363,B 7.7116,C 0.2032,E1 7.8534,E2 420.8347} C_DIS
LIN {X 123.8898,Y 66.9548,Z 174,A 29.4198,B 7.7116,C 0.2055,E1 7.8558,E2 422.6357} C_DIS
LIN {X 125.9731,Y 62.9463,Z 174,A 27.54,B 7.7114,C 0.211,E1 7.8582,E2 424.5219} C_DIS
LIN {X 127.9333,Y 58.8565,Z 174,A 25.9121,B 7.7114,C 0.2115,E1 7.8601,E2 426.123} C_DIS
LIN {X 129.5395,Y 55.2357,Z 174,A 24.0758,B 7.7112,C 0.2202,E1 7.8622,E2 427.9892} C_DIS
LIN {X 131.173,Y 51.2315,Z 174,A 22.5244,B 7.7112,C 0.2207,E1 7.8638,E2 429.515} C_DIS
LIN {X 132.5498,Y 47.5561,Z 174,A 21.0368,B 7.7111,C 0.2228,E1 7.8652,E2 430.9895} C_DIS
LIN {X 133.6985,Y 44.224,Z 174,A 19.6314,B 7.711,C 0.2261,E1 7.8664,E2 432.3922} C_DIS
LIN {X 134.9147,Y 40.3698,Z 174,A 18.0315,B 7.7109,C 0.2297,E1 7.8678,E2 433.9877} C_DIS
LIN {X 135.7504,Y 37.4577,Z 174,A 16.8025,B 7.7108,C 0.2331,E1 7.8687,E2 435.2171} C_DIS
LIN {X 136.5169,Y 34.5566,Z 174,A 15.3878,B 7.7106,C 0.2404,E1 7.8697,E2 436.6575} C_DIS
LIN {X 137.65,Y 29.724,Z 174,A 13.6197,B 7.7106,C 0.241,E1 7.8707,E2 438.3948} C_DIS
LIN {X 138.4227,Y 25.8941,Z 174,A 12.0662,B 7.7104,C 0.2447,E1 7.8716,E2 439.9449} C_DIS
LIN {X 139.093,Y 22.009,Z 174,A 10.4326,B 7.7103,C 0.2499,E1 7.8723,E2 441.5836} C_DIS
LIN {X 139.8564,Y 16.4714,Z 174,A 8.2663,B 7.7101,C 0.2541,E1 7.8731,E2 443.7377} C_DIS
LIN {X 140.1845,Y 13.3934,Z 174,A 6.9409,B 7.71,C 0.2591,E1 7.8735,E2 445.0727} C_DIS
LIN {X 140.4955,Y 9.6185,Z 174,A 5.4567,B 7.7098,C 0.2624,E1 7.8738,E2 446.5509} C_DIS
LIN {X 140.7167,Y 5.469,Z 174,A 3.8165,B 7.7098,C 0.2662,E1 7.874,E2 448.1859} C_DIS
LIN {X 140.8178,Y 1.3772,Z 174,A 2.05,B 7.7095,C 0.2731,E1 7.874,E2 449.9671} C_DIS
LIN {X 140.7749,Y -3.6847,Z 174,A 0.1505,B 7.7094,C 0.2757,E1 7.874,E2 451.8476} C_DIS
LIN {X 140.6302,Y -7.3711,Z 174,A -1.2676,B 7.7093,C 0.2784,E1 7.8738,E2 453.2562} C_DIS
LIN {X 140.3484,Y -11.5547,Z 174,A -3.0833,B 7.709,C 0.2855,E1 7.8734,E2 455.0877} C_DIS
LIN {X 139.9658,Y -15.5194,Z 174,A -4.4952,B 7.709,C 0.2859,E1 7.873,E2 456.474} C_DIS
LIN {X 139.6088,Y -18.4517,Z 174,A -5.7983,B 7.7088,C 0.2914,E1 7.8726,E2 457.7914} C_DIS
LIN {X 139.0713,Y -22.1492,Z 174,A -7.2016,B 7.7088,C 0.2934,E1 7.872,E2 459.181} C_DIS
LIN {X 138.6071,Y -24.8821,Z 174,A -8.2992,B 7.7086,C 0.296,E1 7.8715,E2 460.2756} C_DIS
LIN {X 137.6155,Y -29.8837,Z 174,A -10.3794,B 7.7084,C 0.302,E1 7.8703,E2 462.3585} C_DIS
LIN {X 136.6451,Y -34.0513,Z 174,A -12.2608,B 7.7081,C 0.3098,E1 7.8691,E2 464.2599} C_DIS
LIN {X 134.3737,Y -42.134,Z 174,A -15.3817,B 7.708,C 0.3133,E1 7.8667,E2 467.3457} C_DIS
LIN {X 133.4138,Y -45.0791,Z 174,A -16.6596,B 7.7078,C 0.3171,E1 7.8655,E2 468.6271} C_DIS
LIN {X 132.0306,Y -48.9805,Z 174,A -18.2592,B 7.7077,C 0.32,E1 7.864,E2 470.2173} C_DIS
LIN {X 131.0322,Y -51.5936,Z 174,A -19.3957,B 7.7076,C 0.3231,E1 7.8629,E2 471.3547} C_DIS
LIN {X 129.6421,Y -54.9955,Z 174,A -21.0417,B 7.7073,C 0.3302,E1 7.8611,E2 473.022} C_DIS
LIN {X 127.745,Y -59.2637,Z 174,A -22.8505,B 7.7071,C 0.3334,E1 7.859,E2 474.8206} C_DIS
LIN {X 124.6166,Y -65.5871,Z 174,A -25.2372,B 7.7072,C 0.331,E1 7.8562,E2 477.1467} C_DIS
LIN {X 122.3398,Y -69.7459,Z 174,A -27.5643,B 7.7066,C 0.3441,E1 7.8529,E2 479.5281} C_DIS
LIN {X 120.2192,Y -73.3415,Z 174,A -29.6313,B 7.7061,C 0.3558,E1 7.8499,E2 481.645} C_DIS
LIN {X 117.8567,Y -77.0811,Z 174,A -30.8369,B 7.7065,C 0.3483,E1 7.8481,E2 482.7747} C_DIS
LIN {X 115.9276,Y -79.9525,Z 174,A -32.6129,B 7.706,C 0.3592,E1 7.8453,E2 484.6004} C_DIS
LIN {X 113.9664,Y -82.7235,Z 174,A -34.0539,B 7.7058,C 0.3636,E1 7.8429,E2 486.0506} C_DIS
LIN {X 111.6408,Y -85.8363,Z 174,A -35.4064,B 7.7058,C 0.3628,E1 7.8406,E2 487.3748} C_DIS
LIN {X 108.562,Y -89.6985,Z 174,A -37.3149,B 7.7057,C 0.3654,E1 7.8373,E2 489.272} C_DIS
LIN {X 105.756,Y -92.991,Z 174,A -39.0598,B 7.7055,C 0.369,E1 7.8341,E2 491.0166} C_DIS
LIN {X 102.5028,Y -96.5644,Z 174,A -40.8474,B 7.7055,C 0.3698,E1 7.8308,E2 492.7826} C_DIS
LIN {X 100.5652,Y -98.5806,Z 174,A -42.0543,B 7.7053,C 0.3736,E1 7.8284,E2 493.9997} C_DIS
LIN {X 97.5724,Y -101.5445,Z 174,A -43.8264,B 7.7051,C 0.3783,E1 7.8248,E2 495.7812} C_DIS
LIN {X 94.1337,Y -104.7398,Z 174,A -45.6714,B 7.7049,C 0.3809,E1 7.821,E2 497.6194} C_DIS
LIN {X 91.1817,Y -107.3192,Z 174,A -47.2408,B 7.7048,C 0.3835,E1 7.8177,E2 499.1869} C_DIS
LIN {X 87.8122,Y -110.0934,Z 174,A -48.9487,B 7.7047,C 0.3856,E1 7.814,E2 500.8876} C_DIS
LIN {X 84.7006,Y -112.5049,Z 174,A -50.5651,B 7.7045,C 0.3888,E1 7.8104,E2 502.5073} C_DIS
LIN {X 81.0061,Y -115.1936,Z 174,A -52.5131,B 7.7043,C 0.3938,E1 7.806,E2 504.4687} C_DIS
LIN {X 76.9308,Y -117.9544,Z 174,A -54.4187,B 7.7043,C 0.3953,E1 7.8016,E2 506.3632} C_DIS
LIN {X 73.1453,Y -120.3386,Z 174,A -56.7262,B 7.7036,C 0.4076,E1 7.7959,E2 508.7362} C_DIS
LIN {X 68.6476,Y -122.9601,Z 174,A -58.2416,B 7.704,C 0.3993,E1 7.7924,E2 510.1744} C_DIS
LIN {X 64.9722,Y -124.9394,Z 174,A -59.8812,B 7.704,C 0.4006,E1 7.7884,E2 511.8076} C_DIS
LIN {X 61.1656,Y -126.8463,Z 174,A -61.4795,B 7.704,C 0.4004,E1 7.7844,E2 513.3896} C_DIS
LIN {X 55.1057,Y -129.5957,Z 174,A -64.2865,B 7.7037,C 0.4058,E1 7.7773,E2 516.2121} C_DIS
LIN {X 51.8911,Y -130.9158,Z 174,A -65.6941,B 7.7036,C 0.4074,E1 7.7736,E2 517.6199} C_DIS
LIN {X 48.889,Y -132.0649,Z 174,A -66.9897,B 7.7036,C 0.4086,E1 7.7702,E2 518.9147} C_DIS
LIN {X 44.9345,Y -133.4619,Z 174,A -68.8274,B 7.7033,C 0.4129,E1 7.7653,E2 520.771} C_DIS
LIN {X 40.959,Y -134.7347,Z 174,A -70.3507,B 7.7033,C 0.4113,E1 7.7613,E2 522.2725} C_DIS
LIN {X 37.4525,Y -135.7518,Z 174,A -72.0816,B 7.7031,C 0.4172,E1 7.7566,E2 524.0367} C_DIS
LIN {X 32.4636,Y -137.0308,Z 174,A -73.9809,B 7.7031,C 0.4152,E1 7.7515,E2 525.9116} C_DIS
LIN {X 28.1748,Y -137.9754,Z 174,A -75.7414,B 7.7031,C 0.416,E1 7.7467,E2 527.6698} C_DIS
LIN {X 24.0724,Y -138.752,Z 174,A -77.381,B 7.7031,C 0.416,E1 7.7422,E2 529.3027} C_DIS
LIN {X 20.4743,Y -139.3276,Z 174,A -79.008,B 7.7029,C 0.4195,E1 7.7377,E2 530.9496} C_DIS
LIN {X 16.4324,Y -139.861,Z 174,A -80.5785,B 7.7029,C 0.4187,E1 7.7333,E2 532.5094} C_DIS
LIN {X 12.8235,Y -140.2392,Z 174,A -82.0019,B 7.7029,C 0.4183,E1 7.7294,E2 533.9267} C_DIS
LIN {X 8.8613,Y -140.544,Z 174,A -83.6107,B 7.7029,C 0.4187,E1 7.7249,E2 535.5352} C_DIS
LIN {X 4.6487,Y -140.7481,Z 174,A -85.2893,B 7.7029,C 0.4184,E1 7.7202,E2 537.2099} C_DIS
LIN {X 0.9948,Y -140.8196,Z 174,A -86.8552,B 7.7029,C 0.4201,E1 7.7158,E2 538.7869} C_DIS
Enddeposition()
LIN {X 0.9948,Y -140.8196,Z 174,A -86.8552,B 7.7029,C 0.4201,E1 7.7158,E2 538.7869} C_DIS
Startdeposition()
$VEL.CP = VEL_PRINT
LIN {X 1.7385,Y -141.7208,Z 174,A -85.8274,B 7.7033,C 0.4115,E1 7.7189,E2 537.6955} C_DIS
LIN {X 5.2226,Y -141.6341,Z 174,A -84.3917,B 7.7033,C 0.4107,E1 7.7229,E2 536.2555} C_DIS
LIN {X 9.0918,Y -141.4386,Z 174,A -82.9139,B 7.7033,C 0.4118,E1 7.727,E2 534.7888} C_DIS
LIN {X 12.1677,Y -141.2069,Z 174,A -81.6653,B 7.7033,C 0.4114,E1 7.7304,E2 533.5392} C_DIS
LIN {X 15.6229,Y -140.867,Z 174,A -80.2572,B 7.7033,C 0.4107,E1 7.7344,E2 532.1298} C_DIS
LIN {X 19.1065,Y -140.4379,Z 174,A -78.8575,B 7.7033,C 0.4104,E1 7.7382,E2 530.7319} C_DIS
LIN {X 22.5379,Y -139.9287,Z 174,A -77.3345,B 7.7036,C 0.4073,E1 7.7425,E2 529.1919} C_DIS
LIN {X 26.5946,Y -139.2123,Z 174,A -75.8412,B 7.7034,C 0.4095,E1 7.7465,E2 527.7205} C_DIS
LIN {X 29.7377,Y -138.575,Z 174,A -74.4973,B 7.7035,C 0.4077,E1 7.7502,E2 526.3694} C_DIS
LIN {X 33.1179,Y -137.8062,Z 174,A -73.2004,B 7.7035,C 0.4086,E1 7.7537,E2 525.0857} C_DIS
LIN {X 36.099,Y -137.0561,Z 174,A -71.8272,B 7.7037,C 0.4051,E1 7.7575,E2 523.6941} C_DIS
LIN {X 39.8533,Y -136.0111,Z 174,A -70.3868,B 7.7037,C 0.4062,E1 7.7613,E2 522.2707} C_DIS
LIN {X 42.8279,Y -135.1043,Z 174,A -69.0525,B 7.7037,C 0.4035,E1 7.7649,E2 520.9252} C_DIS
LIN {X 46.1247,Y -134.0146,Z 174,A -67.6591,B 7.7038,C 0.4023,E1 7.7686,E2 519.5322} C_DIS
LIN {X 49.7571,Y -132.7084,Z 174,A -66.0678,B 7.7039,C 0.3999,E1 7.7728,E2 517.9355} C_DIS
LIN {X 52.9925,Y -131.4499,Z 174,A -64.7005,B 7.7039,C 0.399,E1 7.7763,E2 516.572} C_DIS
LIN {X 55.8756,Y -130.2511,Z 174,A -63.4696,B 7.704,C 0.398,E1 7.7794,E2 515.3443} C_DIS
LIN {X 59.0337,Y -128.8508,Z 174,A -62.087,B 7.7041,C 0.3965,E1 7.783,E2 513.9625} C_DIS
LIN {X 62.3298,Y -127.2887,Z 174,A -60.6766,B 7.7041,C 0.3958,E1 7.7865,E2 512.5595} C_DIS
LIN {X 65.2738,Y -125.8057,Z 174,A -59.3145,B 7.7043,C 0.3933,E1 7.7899,E2 511.1924} C_DIS
LIN {X 68.5501,Y -124.0513,Z 174,A -57.7315,B 7.7045,C 0.3895,E1 7.7938,E2 509.5973} C_DIS
LIN {X 72.3124,Y -121.8968,Z 174,A -55.9571,B 7.7046,C 0.3864,E1 7.7981,E2 507.8186} C_DIS
LIN {X 76.4049,Y -119.3739,Z 174,A -54.093,B 7.7047,C 0.3848,E1 7.8025,E2 505.9634} C_DIS
LIN {X 80.0542,Y -116.9581,Z 174,A -52.3682,B 7.7048,C 0.3826,E1 7.8065,E2 504.243} C_DIS
LIN {X 83.5833,Y -114.4632,Z 174,A -50.6332,B 7.705,C 0.3798,E1 7.8104,E2 502.5081} C_DIS
LIN {X 87.0491,Y -111.8497,Z 174,A -48.9128,B 7.705,C 0.3772,E1 7.8142,E2 500.7908} C_DIS
LIN {X 90.0647,Y -109.4365,Z 174,A -47.2689,B 7.7053,C 0.3726,E1 7.8178,E2 499.1343} C_DIS
LIN {X 93.7499,Y -106.2958,Z 174,A -45.3965,B 7.7054,C 0.3705,E1 7.8217,E2 497.2716} C_DIS
LIN {X 97.1042,Y -103.2407,Z 174,A -43.619,B 7.7055,C 0.3679,E1 7.8254,E2 495.4999} C_DIS
LIN {X 100.2201,Y -100.2195,Z 174,A -41.7935,B 7.7058,C 0.3628,E1 7.829,E2 493.6632} C_DIS
LIN {X 103.3937,Y -96.942,Z 174,A -39.9752,B 7.7059,C 0.3593,E1 7.8325,E2 491.8467} C_DIS
LIN {X 106.314,Y -93.7294,Z 174,A -38.2578,B 7.7061,C 0.3562,E1 7.8357,E2 490.1326} C_DIS
LIN {X 109.4372,Y -90.064,Z 174,A -36.3428,B 7.7063,C 0.3524,E1 7.8391,E2 488.2199} C_DIS
LIN {X 112.2986,Y -86.4699,Z 174,A -34.5894,B 7.7063,C 0.3502,E1 7.8421,E2 486.4787} C_DIS
LIN {X 114.8899,Y -82.9951,Z 174,A -32.8766,B 7.7065,C 0.3468,E1 7.845,E2 484.7694} C_DIS
LIN {X 117.3663,Y -79.4543,Z 174,A -31.1532,B 7.7067,C 0.3431,E1 7.8477,E2 483.0474} C_DIS
LIN {X 119.7317,Y -75.8432,Z 174,A -29.4244,B 7.7068,C 0.3391,E1 7.8503,E2 481.319} C_DIS
LIN {X 121.9126,Y -72.286,Z 174,A -27.7362,B 7.707,C 0.3348,E1 7.8527,E2 479.629} C_DIS
LIN {X 124.1686,Y -68.3382,Z 174,A -25.9243,B 7.7072,C 0.3306,E1 7.8552,E2 477.8188} C_DIS
LIN {X 125.9253,Y -65.0444,Z 174,A -24.3934,B 7.7074,C 0.3263,E1 7.8572,E2 476.2834} C_DIS
LIN {X 127.8378,Y -61.1945,Z 174,A -22.8529,B 7.7074,C 0.3258,E1 7.8591,E2 474.7675} C_DIS
LIN {X 129.3012,Y -58.0387,Z 174,A -21.6637,B 7.7074,C 0.3265,E1 7.8604,E2 473.6058} C_DIS
LIN {X 130.2684,Y -55.8356,Z 174,A -20.468,B 7.7077,C 0.3193,E1 7.8618,E2 472.3794} C_DIS
LIN {X 131.7875,Y -52.1544,Z 174,A -18.6933,B 7.708,C 0.3115,E1 7.8636,E2 470.5812} C_DIS
LIN {X 133.5792,Y -47.3755,Z 174,A -16.8604,B 7.708,C 0.3107,E1 7.8654,E2 468.777} C_DIS
LIN {X 134.7008,Y -44.0853,Z 174,A -15.4807,B 7.7082,C 0.3073,E1 7.8666,E2 467.3994} C_DIS
LIN {X 135.6449,Y -41.0844,Z 174,A -14.234,B 7.7082,C 0.3043,E1 7.8676,E2 466.1547} C_DIS
LIN {X 136.7093,Y -37.3968,Z 174,A -12.7126,B 7.7084,C 0.3006,E1 7.8688,E2 464.6359} C_DIS
LIN {X 137.4899,Y -34.4103,Z 174,A -11.4877,B 7.7085,C 0.2976,E1 7.8696,E2 463.4128} C_DIS
LIN {X 138.3878,Y -30.6049,Z 174,A -9.8189,B 7.7088,C 0.2913,E1 7.8707,E2 461.7308} C_DIS
LIN {X 139.0868,Y -27.2511,Z 174,A -8.6484,B 7.7088,C 0.2918,E1 7.8713,E2 460.5874} C_DIS
LIN {X 139.7126,Y -23.8331,Z 174,A -7.1862,B 7.709,C 0.2866,E1 7.872,E2 459.1162} C_DIS
LIN {X 140.2542,Y -20.4023,Z 174,A -5.8103,B 7.709,C 0.2832,E1 7.8726,E2 457.7428} C_DIS
LIN {X 140.7116,Y -16.9604,Z 174,A -4.4351,B 7.7092,C 0.2797,E1 7.8731,E2 456.37} C_DIS
LIN {X 141.0847,Y -13.5088,Z 174,A -3.1297,B 7.7092,C 0.2777,E1 7.8734,E2 455.0763} C_DIS
LIN {X 141.3472,Y -10.4101,Z 174,A -1.8258,B 7.7094,C 0.2731,E1 7.8737,E2 453.7651} C_DIS
LIN {X 141.5794,Y -6.5571,Z 174,A -0.3352,B 7.7096,C 0.2701,E1 7.8739,E2 452.2824} C_DIS
LIN {X 141.6998,Y -2.9978,Z 174,A 1.2378,B 7.7098,C 0.2632,E1 7.874,E2 450.6905} C_DIS
LIN {X 141.7255,Y 1.2994,Z 174,A 2.9181,B 7.7099,C 0.2593,E1 7.874,E2 449.0162} C_DIS
LIN {X 141.6338,Y 5.2304,Z 174,A 4.4543,B 7.71,C 0.2559,E1 7.874,E2 447.4857} C_DIS
LIN {X 141.3932,Y 9.7809,Z 174,A 6.0767,B 7.71,C 0.2552,E1 7.8736,E2 445.8907} C_DIS
LIN {X 141.2076,Y 12.1596,Z 174,A 7.132,B 7.7102,C 0.2505,E1 7.8734,E2 444.8226} C_DIS
LIN {X 140.863,Y 15.66,Z 174,A 8.523,B 7.7103,C 0.2471,E1 7.873,E2 443.4346} C_DIS
LIN {X 140.4387,Y 19.1001,Z 174,A 9.8968,B 7.7104,C 0.2436,E1 7.8725,E2 442.0633} C_DIS
LIN {X 139.9303,Y 22.5285,Z 174,A 11.4365,B 7.7106,C 0.2368,E1 7.8718,E2 440.5042} C_DIS
LIN {X 139.3368,Y 25.9436,Z 174,A 12.7621,B 7.7107,C 0.2344,E1 7.8712,E2 439.1875} C_DIS
LIN {X 138.5781,Y 29.7237,Z 174,A 14.1921,B 7.7107,C 0.2327,E1 7.8704,E2 437.7731} C_DIS
LIN {X 137.8095,Y 33.104,Z 174,A 15.4701,B 7.7108,C 0.2313,E1 7.8696,E2 436.5104} C_DIS
LIN {X 137.0506,Y 36.1197,Z 174,A 16.8039,B 7.711,C 0.2262,E1 7.8686,E2 435.1656} C_DIS
LIN {X 136.1198,Y 39.482,Z 174,A 18.1883,B 7.711,C 0.2229,E1 7.8676,E2 433.7836} C_DIS
LIN {X 135.1109,Y 42.8074,Z 174,A 19.5675,B 7.7112,C 0.2195,E1 7.8664,E2 432.4068} C_DIS
LIN {X 134.0208,Y 46.1069,Z 174,A 20.9465,B 7.7112,C 0.2162,E1 7.8652,E2 431.0302} C_DIS
LIN {X 132.7102,Y 49.7523,Z 174,A 22.5612,B 7.7114,C 0.211,E1 7.8636,E2 429.4081} C_DIS
LIN {X 130.9329,Y 54.2586,Z 174,A 24.4067,B 7.7114,C 0.2081,E1 7.8617,E2 427.5761} C_DIS
LIN {X 129.5687,Y 57.4406,Z 174,A 25.8411,B 7.7116,C 0.2037,E1 7.8601,E2 426.1363} C_DIS
LIN {X 128.1273,Y 60.5885,Z 174,A 27.2548,B 7.7116,C 0.1998,E1 7.8584,E2 424.72} C_DIS
LIN {X 126.2912,Y 64.3256,Z 174,A 28.62,B 7.7116,C 0.202,E1 7.8568,E2 423.3953} C_DIS
LIN {X 124.6789,Y 67.4028,Z 174,A 30.2375,B 7.7118,C 0.1941,E1 7.8546,E2 421.7493} C_DIS
LIN {X 122.5438,Y 71.2102,Z 174,A 31.9983,B 7.7119,C 0.1898,E1 7.8522,E2 419.9881} C_DIS
LIN {X 120.2031,Y 75.0939,Z 174,A 33.8618,B 7.7121,C 0.1847,E1 7.8495,E2 418.1197} C_DIS
LIN {X 117.8487,Y 78.737,Z 174,A 35.5823,B 7.7121,C 0.1812,E1 7.8468,E2 416.4027} C_DIS
LIN {X 115.3731,Y 82.3219,Z 174,A 37.3059,B 7.7122,C 0.1778,E1 7.8441,E2 414.6832} C_DIS
LIN {X 112.6991,Y 85.9464,Z 174,A 39.104,B 7.7123,C 0.1741,E1 7.8411,E2 412.8873} C_DIS
LIN {X 109.89,Y 89.5101,Z 174,A 40.9107,B 7.7123,C 0.1706,E1 7.8379,E2 411.0834} C_DIS
LIN {X 106.8708,Y 93.0939,Z 174,A 42.707,B 7.7124,C 0.1684,E1 7.8347,E2 409.2993} C_DIS
LIN {X 104.2886,Y 95.9777,Z 174,A 44.2812,B 7.7125,C 0.1649,E1 7.8317,E2 407.7233} C_DIS
LIN {X 101.3018,Y 99.1252,Z 174,A 46.0261,B 7.7125,C 0.1614,E1 7.8283,E2 405.9791} C_DIS
LIN {X 98.2644,Y 102.1378,Z 174,A 47.6887,B 7.7126,C 0.1593,E1 7.825,E2 404.3247} C_DIS
LIN {X 95.106,Y 105.0842,Z 174,A 49.3985,B 7.7126,C 0.1566,E1 7.8215,E2 402.6191} C_DIS
LIN {X 92.3051,Y 107.553,Z 174,A 50.9586,B 7.7128,C 0.1528,E1 7.8182,E2 401.0522} C_DIS
LIN {X 89.0827,Y 110.2366,Z 174,A 52.6468,B 7.7128,C 0.1499,E1 7.8146,E2 399.3646} C_DIS
LIN {X 85.6628,Y 112.9152,Z 174,A 54.402,B 7.7128,C 0.1468,E1 7.8107,E2 397.6091} C_DIS
LIN {X 82.1614,Y 115.4879,Z 174,A 56.0215,B 7.7128,C 0.1465,E1 7.807,E2 396.0071} C_DIS
LIN {X 79.2941,Y 117.4747,Z 174,A 57.5299,B 7.713,C 0.1424,E1 7.8035,E2 394.4859} C_DIS
LIN {X 75.6609,Y 119.8468,Z 174,A 59.1452,B 7.713,C 0.1423,E1 7.7998,E2 392.8883} C_DIS
LIN {X 72.2474,Y 121.9356,Z 174,A 60.8175,B 7.713,C 0.1389,E1 7.7958,E2 391.2089} C_DIS
LIN {X 68.3382,Y 124.1686,Z 174,A 62.5961,B 7.713,C 0.1371,E1 7.7914,E2 389.4357} C_DIS
LIN {X 65.078,Y 125.9082,Z 174,A 64.1627,B 7.7131,C 0.1338,E1 7.7875,E2 387.8596} C_DIS
LIN {X 61.3656,Y 127.7561,Z 174,A 65.6909,B 7.7131,C 0.1344,E1 7.7838,E2 386.3505} C_DIS
LIN {X 58.0476,Y 129.2972,Z 174,A 66.9244,B 7.7131,C 0.1372,E1 7.7807,E2 385.1487} C_DIS
LIN {X 55.1766,Y 130.5495,Z 174,A 68.5589,B 7.7131,C 0.129,E1 7.7764,E2 383.4668} C_DIS
LIN {X 50.7056,Y 132.3507,Z 174,A 70.5149,B 7.7132,C 0.1268,E1 7.7713,E2 381.5102} C_DIS
LIN {X 47.3767,Y 133.5787,Z 174,A 71.7812,B 7.7132,C 0.1285,E1 7.768,E2 380.2657} C_DIS
LIN {X 44.0864,Y 134.7005,Z 174,A 73.1765,B 7.7132,C 0.1274,E1 7.7643,E2 378.872} C_DIS
LIN {X 41.1458,Y 135.6261,Z 174,A 74.4153,B 7.7132,C 0.1265,E1 7.761,E2 377.6343} C_DIS
LIN {X 37.3255,Y 136.729,Z 174,A 76.1349,B 7.7132,C 0.1232,E1 7.7564,E2 375.9006} C_DIS
LIN {X 33.1015,Y 137.8101,Z 174,A 77.8159,B 7.7132,C 0.1235,E1 7.7518,E2 374.2304} C_DIS
LIN {X 29.3362,Y 138.6617,Z 174,A 79.3852,B 7.7132,C 0.1224,E1 7.7476,E2 372.6605} C_DIS
LIN {X 25.9375,Y 139.338,Z 174,A 80.8054,B 7.7133,C 0.1213,E1 7.7437,E2 371.2383} C_DIS
LIN {X 22.1188,Y 139.994,Z 174,A 82.2885,B 7.7133,C 0.122,E1 7.7396,E2 369.7663} C_DIS
LIN {X 18.6832,Y 140.4934,Z 174,A 83.6886,B 7.7133,C 0.1215,E1 7.7357,E2 368.367} C_DIS
LIN {X 15.2235,Y 140.91,Z 174,A 85.0876,B 7.7133,C 0.1212,E1 7.7318,E2 366.9697} C_DIS
LIN {X 12.1555,Y 141.208,Z 174,A 86.3355,B 7.7133,C 0.1209,E1 7.7284,E2 365.7221} C_DIS
LIN {X 8.6939,Y 141.4631,Z 174,A 87.7346,B 7.7133,C 0.1207,E1 7.7245,E2 364.3241} C_DIS
LIN {X 5.1983,Y 141.6351,Z 174,A 89.1806,B 7.7133,C 0.12,E1 7.7204,E2 362.8747} C_DIS
LIN {X 1.3396,Y 141.7249,Z 174,A 90.5992,B 7.7133,C 0.1224,E1 7.7165,E2 361.475} C_DIS
LIN {X -1.7439,Y 141.7207,Z 174,A 91.9719,B 7.7133,C 0.1202,E1 7.7127,E2 360.0867} C_DIS
LIN {X -6.0836,Y 141.6006,Z 174,A 93.6639,B 7.7133,C 0.1215,E1 7.708,E2 358.4036} C_DIS
LIN {X -9.0864,Y 141.439,Z 174,A 94.9175,B 7.7133,C 0.121,E1 7.7044,E2 357.1458} C_DIS
LIN {X -12.1778,Y 141.2061,Z 174,A 96.1757,B 7.7133,C 0.1213,E1 7.7009,E2 355.8875} C_DIS
LIN {X -15.6306,Y 140.8662,Z 174,A 97.5776,B 7.7133,C 0.1217,E1 7.6971,E2 354.4865} C_DIS
LIN {X -19.0745,Y 140.4421,Z 174,A 98.9881,B 7.7133,C 0.1221,E1 7.6931,E2 353.0758} C_DIS
LIN {X -22.5962,Y 139.919,Z 174,A 100.5472,B 7.7133,C 0.1207,E1 7.6888,E2 351.5022} C_DIS
LIN {X -26.0162,Y 139.3229,Z 174,A 101.9424,B 7.7133,C 0.1216,E1 7.685,E2 350.1089} C_DIS
LIN {X -29.7728,Y 138.5674,Z 174,A 103.4436,B 7.7133,C 0.1233,E1 7.6809,E2 348.6148} C_DIS
LIN {X -33.1223,Y 137.8051,Z 174,A 104.7886,B 7.7133,C 0.1249,E1 7.6772,E2 347.2762} C_DIS
LIN {X -36.1326,Y 137.0471,Z 174,A 106.0593,B 7.7133,C 0.1256,E1 7.6738,E2 346.0043} C_DIS
LIN {X -39.8561,Y 136.0103,Z 174,A 107.5422,B 7.7132,C 0.1281,E1 7.6699,E2 344.5326} C_DIS
LIN {X -42.8057,Y 135.1114,Z 174,A 108.8822,B 7.7132,C 0.1277,E1 7.6663,E2 343.1815} C_DIS
LIN {X -46.1515,Y 134.0053,Z 174,A 110.3142,B 7.7132,C 0.1289,E1 7.6625,E2 341.7496} C_DIS
LIN {X -49.7757,Y 132.7014,Z 174,A 111.8823,B 7.7132,C 0.1303,E1 7.6584,E2 340.1811} C_DIS
LIN {X -53.0052,Y 131.4447,Z 174,A 113.38,B 7.7132,C 0.1303,E1 7.6544,E2 338.6721} C_DIS
LIN {X -57.4298,Y 129.5736,Z 174,A 115.2448,B 7.7132,C 0.1337,E1 7.6497,E2 336.8187} C_DIS
LIN {X -60.6631,Y 128.0917,Z 174,A 116.732,B 7.7131,C 0.1347,E1 7.6459,E2 335.3263} C_DIS
LIN {X -63.73,Y 126.5944,Z 174,A 118.0843,B 7.7131,C 0.1369,E1 7.6425,E2 333.9787} C_DIS
LIN {X -66.8134,Y 124.9956,Z 174,A 119.5534,B 7.7131,C 0.1377,E1 7.6389,E2 332.5023} C_DIS
LIN {X -70.6247,Y 122.8827,Z 174,A 121.3305,B 7.713,C 0.14,E1 7.6346,E2 330.7247} C_DIS
LIN {X -74.351,Y 120.6642,Z 174,A 123.1846,B 7.713,C 0.1411,E1 7.6301,E2 328.8591} C_DIS
LIN {X -78.0068,Y 118.3333,Z 174,A 124.9504,B 7.713,C 0.1436,E1 7.626,E2 327.0931} C_DIS
LIN {X -81.6695,Y 115.8357,Z 174,A 126.7511,B 7.7129,C 0.1465,E1 7.6218,E2 325.2929} C_DIS
LIN {X -85.1835,Y 113.2769,Z 174,A 128.5322,B 7.7129,C 0.1491,E1 7.6178,E2 323.5103} C_DIS
LIN {X -88.585,Y 110.6376,Z 174,A 130.212,B 7.7127,C 0.1532,E1 7.6142,E2 321.8399} C_DIS
LIN {X -91.9074,Y 107.8929,Z 174,A 131.9561,B 7.7127,C 0.1564,E1 7.6105,E2 320.097} C_DIS
LIN {X -95.0676,Y 105.1191,Z 174,A 133.7039,B 7.7127,C 0.159,E1 7.6068,E2 318.3447} C_DIS
LIN {X -97.8915,Y 102.4943,Z 174,A 135.3535,B 7.7126,C 0.1607,E1 7.6034,E2 316.6848} C_DIS
LIN {X -100.8361,Y 99.5996,Z 174,A 136.9551,B 7.7125,C 0.1651,E1 7.6003,E2 315.0935} C_DIS
LIN {X -103.4533,Y 96.8782,Z 174,A 138.6189,B 7.7125,C 0.1663,E1 7.5971,E2 313.4134} C_DIS
LIN {X -106.3759,Y 93.6593,Z 174,A 140.3944,B 7.7124,C 0.1698,E1 7.5938,E2 311.6373} C_DIS
LIN {X -109.4621,Y 90.0337,Z 174,A 142.2987,B 7.7123,C 0.1744,E1 7.5903,E2 309.7374} C_DIS
LIN {X -112.2297,Y 86.5588,Z 174,A 144.0882,B 7.7123,C 0.1786,E1 7.5873,E2 307.9505} C_DIS
LIN {X -114.4724,Y 83.5707,Z 174,A 145.7137,B 7.7122,C 0.1804,E1 7.5846,E2 306.3116} C_DIS
LIN {X -116.9777,Y 80.0256,Z 174,A 147.3661,B 7.712,C 0.1861,E1 7.5819,E2 304.6742} C_DIS
LIN {X -118.9258,Y 77.1005,Z 174,A 148.9237,B 7.712,C 0.1875,E1 7.5795,E2 303.1002} C_DIS
LIN {X -121.4707,Y 73.0263,Z 174,A 150.857,B 7.7119,C 0.1925,E1 7.5767,E2 301.17} C_DIS
LIN {X -123.7488,Y 69.0957,Z 174,A 152.6853,B 7.7118,C 0.1972,E1 7.5742,E2 299.3445} C_DIS
LIN {X -125.8061,Y 65.2729,Z 174,A 154.5746,B 7.7117,C 0.1997,E1 7.5717,E2 297.4396} C_DIS
LIN {X -127.6603,Y 61.566,Z 174,A 156.2493,B 7.7116,C 0.2041,E1 7.5697,E2 295.7667} C_DIS
LIN {X -129.382,Y 57.858,Z 174,A 157.8149,B 7.7114,C 0.2097,E1 7.5679,E2 294.2139} C_DIS
LIN {X -131.1318,Y 53.7817,Z 174,A 159.6407,B 7.7114,C 0.2141,E1 7.5659,E2 292.3858} C_DIS
LIN {X -132.2388,Y 50.9933,Z 174,A 160.8809,B 7.7112,C 0.2169,E1 7.5646,E2 291.1431} C_DIS
LIN {X -133.58,Y 47.3732,Z 174,A 162.4703,B 7.7112,C 0.2208,E1 7.5631,E2 289.5516} C_DIS
LIN {X -134.7011,Y 44.0845,Z 174,A 163.8991,B 7.711,C 0.2243,E1 7.5618,E2 288.121} C_DIS
LIN {X -135.6267,Y 41.1441,Z 174,A 165.1678,B 7.711,C 0.2274,E1 7.5608,E2 286.8505} C_DIS
LIN {X -136.7002,Y 37.4295,Z 174,A 166.7578,B 7.7108,C 0.2314,E1 7.5596,E2 285.2587} C_DIS
LIN {X -137.6986,Y 33.5643,Z 174,A 168.4978,B 7.7108,C 0.2341,E1 7.5584,E2 283.5038} C_DIS
LIN {X -138.6744,Y 29.2772,Z 174,A 170.2894,B 7.7106,C 0.2389,E1 7.5573,E2 281.7121} C_DIS
LIN {X -139.3492,Y 25.8785,Z 174,A 171.742,B 7.7105,C 0.2421,E1 7.5566,E2 280.2541} C_DIS
LIN {X -140.0031,Y 22.0596,Z 174,A 173.2368,B 7.7103,C 0.2476,E1 7.5559,E2 278.77} C_DIS
LIN {X -140.4945,Y 18.6747,Z 174,A 174.6514,B 7.7102,C 0.2511,E1 7.5553,E2 277.3525} C_DIS
LIN {X -140.9142,Y 15.1848,Z 174,A 176.0977,B 7.7101,C 0.2548,E1 7.5549,E2 275.9042} C_DIS
LIN {X -141.2117,Y 12.1108,Z 174,A 177.3737,B 7.71,C 0.258,E1 7.5546,E2 274.6258} C_DIS
LIN {X -141.4654,Y 8.6569,Z 174,A 178.8395,B 7.7099,C 0.2611,E1 7.5543,E2 273.1526} C_DIS
LIN {X -141.6349,Y 5.2037,Z 174,A -179.7444,B 7.7097,C 0.2649,E1 7.5541,E2 271.7354} C_DIS
LIN {X -141.7266,Y 1.1435,Z 174,A -178.333,B 7.7095,C 0.2729,E1 7.5541,E2 270.3555} C_DIS
LIN {X -141.72,Y -1.7853,Z 174,A -176.8788,B 7.7095,C 0.2724,E1 7.5541,E2 268.8671} C_DIS
LIN {X -141.633,Y -5.2518,Z 174,A -175.396,B 7.7094,C 0.2753,E1 7.5542,E2 267.3749} C_DIS
LIN {X -141.4387,Y -9.0904,Z 174,A -173.8944,B 7.7092,C 0.2805,E1 7.5545,E2 265.8814} C_DIS
LIN {X -141.2085,Y -12.1497,Z 174,A -172.6255,B 7.7091,C 0.2837,E1 7.5548,E2 264.6098} C_DIS
LIN {X -140.8705,Y -15.5907,Z 174,A -171.2037,B 7.7089,C 0.2873,E1 7.5552,E2 263.1861} C_DIS
LIN {X -140.4478,Y -19.0305,Z 174,A -169.7757,B 7.7089,C 0.2909,E1 7.5557,E2 261.7557} C_DIS
LIN {X -139.933,Y -22.5115,Z 174,A -168.1811,B 7.7087,C 0.2925,E1 7.5564,E2 260.1397} C_DIS
LIN {X -139.3362,Y -25.9467,Z 174,A -166.7726,B 7.7086,C 0.2965,E1 7.5571,E2 258.7325} C_DIS
LIN {X -138.5748,Y -29.7385,Z 174,A -165.2845,B 7.7084,C 0.3019,E1 7.5579,E2 257.2553} C_DIS
LIN {X -137.8039,Y -33.1274,Z 174,A -163.9521,B 7.7082,C 0.3069,E1 7.5588,E2 255.9335} C_DIS
LIN {X -137.0464,Y -36.1352,Z 174,A -162.5759,B 7.7082,C 0.3086,E1 7.5597,E2 254.5422} C_DIS
LIN {X -135.9402,Y -40.0955,Z 174,A -160.7899,B 7.708,C 0.3114,E1 7.5611,E2 252.7411} C_DIS
LIN {X -134.577,Y -44.4573,Z 174,A -159.0038,B 7.7078,C 0.3173,E1 7.5626,E2 250.9644} C_DIS
LIN {X -133.4415,Y -47.7575,Z 174,A -157.4871,B 7.7077,C 0.3195,E1 7.5641,E2 249.4348} C_DIS
LIN {X -132.0923,Y -51.3702,Z 174,A -155.9805,B 7.7075,C 0.3244,E1 7.5655,E2 247.936} C_DIS
LIN {X -130.7959,Y -54.5867,Z 174,A -154.4709,B 7.7074,C 0.3265,E1 7.5672,E2 246.4131} C_DIS
LIN {X -128.8542,Y -59.0264,Z 174,A -152.5647,B 7.7071,C 0.3324,E1 7.5693,E2 244.5151} C_DIS
LIN {X -127.2823,Y -62.3428,Z 174,A -150.951,B 7.7071,C 0.3343,E1 7.5713,E2 242.8851} C_DIS
LIN {X -125.807,Y -65.2712,Z 174,A -149.7102,B 7.7069,C 0.3389,E1 7.5729,E2 241.6563} C_DIS
LIN {X -124.0539,Y -68.5454,Z 174,A -148.0683,B 7.7068,C 0.3405,E1 7.5751,E2 239.9968} C_DIS
LIN {X -121.9044,Y -72.2996,Z 174,A -146.2774,B 7.7066,C 0.3442,E1 7.5776,E2 238.2012} C_DIS
LIN {X -119.3761,Y -76.4014,Z 174,A -144.385,B 7.7064,C 0.3497,E1 7.5804,E2 236.3171} C_DIS
LIN {X -116.9792,Y -80.0234,Z 174,A -142.5975,B 7.7062,C 0.3533,E1 7.5832,E2 234.5263} C_DIS
LIN {X -114.4726,Y -83.5704,Z 174,A -140.8107,B 7.706,C 0.3568,E1 7.5861,E2 232.7361} C_DIS
LIN {X -111.858,Y -87.0384,Z 174,A -139.0424,B 7.7059,C 0.3605,E1 7.5891,E2 230.9669} C_DIS
LIN {X -109.4361,Y -90.0652,Z 174,A -137.3465,B 7.7059,C 0.362,E1 7.5921,E2 229.2546} C_DIS
LIN {X -106.2907,Y -93.7557,Z 174,A -135.4229,B 7.7056,C 0.3667,E1 7.5957,E2 227.3365} C_DIS
LIN {X -103.2411,Y -97.1037,Z 174,A -133.8095,B 7.7052,C 0.3738,E1 7.5987,E2 225.7525} C_DIS
LIN {X -101.0684,Y -99.3631,Z 174,A -132.306,B 7.7053,C 0.3726,E1 7.6016,E2 224.2181} C_DIS
LIN {X -97.8863,Y -102.4993,Z 174,A -130.4874,B 7.7051,C 0.3759,E1 7.6053,E2 222.3984} C_DIS
LIN {X -94.6749,Y -105.4728,Z 174,A -128.6611,B 7.7051,C 0.3783,E1 7.6091,E2 220.5649} C_DIS
LIN {X -91.2463,Y -108.4526,Z 174,A -126.761,B 7.7049,C 0.3806,E1 7.6131,E2 218.6567} C_DIS
LIN {X -87.7266,Y -111.319,Z 174,A -124.902,B 7.7048,C 0.3834,E1 7.6172,E2 216.7949} C_DIS
LIN {X -84.2743,Y -113.9556,Z 174,A -123.2349,B 7.7046,C 0.3877,E1 7.6209,E2 215.1399} C_DIS
LIN {X -80.8904,Y -116.3812,Z 174,A -121.5099,B 7.7045,C 0.3897,E1 7.6248,E2 213.4095} C_DIS
LIN {X -77.2933,Y -118.8006,Z 174,A -119.7252,B 7.7044,C 0.3918,E1 7.629,E2 211.6206} C_DIS
LIN {X -74.1791,Y -120.7696,Z 174,A -118.1905,B 7.7043,C 0.3932,E1 7.6326,E2 210.08} C_DIS
LIN {X -70.4429,Y -122.9865,Z 174,A -116.4026,B 7.7042,C 0.395,E1 7.637,E2 208.288} C_DIS
LIN {X -66.6169,Y -125.1004,Z 174,A -114.7249,B 7.704,C 0.3987,E1 7.6411,E2 206.6223} C_DIS
LIN {X -63.108,Y -126.9049,Z 174,A -113.0212,B 7.704,C 0.3988,E1 7.6453,E2 204.9039} C_DIS
LIN {X -59.6362,Y -128.5722,Z 174,A -111.5364,B 7.7038,C 0.4018,E1 7.6491,E2 203.4286} C_DIS
LIN {X -57.0745,Y -129.7325,Z 174,A -110.3892,B 7.7038,C 0.4028,E1 7.652,E2 202.2801} C_DIS
LIN {X -53.6575,Y -131.1818,Z 174,A -108.7141,B 7.7038,C 0.4014,E1 7.6564,E2 200.5815} C_DIS
LIN {X -49.3788,Y -132.8501,Z 174,A -106.9794,B 7.7037,C 0.4052,E1 7.6609,E2 198.8629} C_DIS
LIN {X -45.7371,Y -134.1489,Z 174,A -105.4423,B 7.7036,C 0.4069,E1 7.6649,E2 197.329} C_DIS
LIN {X -42.4341,Y -135.2301,Z 174,A -103.9666,B 7.7036,C 0.4068,E1 7.6689,E2 195.8436} C_DIS
LIN {X -38.9788,Y -136.2669,Z 174,A -102.5764,B 7.7035,C 0.409,E1 7.6726,E2 194.4622} C_DIS
LIN {X -35.7282,Y -137.1549,Z 174,A -101.2066,B 7.7035,C 0.4097,E1 7.6763,E2 193.0911} C_DIS
LIN {X -32.7316,Y -137.8993,Z 174,A -99.9497,B 7.7035,C 0.4102,E1 7.6797,E2 191.8326} C_DIS
LIN {X -29.3487,Y -138.659,Z 174,A -98.4795,B 7.7035,C 0.4097,E1 7.6837,E2 190.3529} C_DIS
LIN {X -25.8206,Y -139.3603,Z 174,A -96.9979,B 7.7035,C 0.4099,E1 7.6878,E2 188.8673} C_DIS
LIN {X -22.1256,Y -139.9929,Z 174,A -95.5524,B 7.7033,C 0.4116,E1 7.6918,E2 187.4306} C_DIS
LIN {X -18.6782,Y -140.494,Z 174,A -94.1464,B 7.7033,C 0.4121,E1 7.6956,E2 186.0243} C_DIS
LIN {X -15.2295,Y -140.9094,Z 174,A -92.7442,B 7.7033,C 0.4124,E1 7.6995,E2 184.6219} C_DIS
LIN {X -12.1619,Y -141.2074,Z 174,A -91.4886,B 7.7033,C 0.4124,E1 7.703,E2 183.3646} C_DIS
LIN {X -8.675,Y -141.4643,Z 174,A -90.0405,B 7.7033,C 0.4119,E1 7.7071,E2 181.9113} C_DIS
LIN {X -4.1809,Y -141.6686,Z 174,A -88.4542,B 7.7031,C 0.416,E1 7.7114,E2 180.3553} C_DIS
LIN {X -1.3447,Y -141.7249,Z 174,A -87.2249,B 7.7031,C 0.4145,E1 7.7149,E2 179.1145} C_DIS
LIN {X 1.0008,Y -141.7257,Z 174,A -86.5041,B 7.703,C 0.4184,E1 7.7168,E2 178.4236} C_DIS
Enddeposition()
LIN {X 0.9619,Y -132.7934,Z 175,A -86.8622,B 7.893,C 0.377,E1 7.9045,E2 178.4349} C_DIS
Startdeposition()
$VEL.CP = VEL_PRINT
LIN {X -1.6481,Y -132.7885,Z 175,A -88.1906,B 7.8929,C 0.3806,E1 7.9008,E2 179.7888} C_DIS
LIN {X -4.588,Y -132.7195,Z 175,A -89.5662,B 7.8928,C 0.3825,E1 7.8969,E2 181.1782} C_DIS
LIN {X -8.1493,Y -132.5472,Z 175,A -91.022,B 7.8928,C 0.381,E1 7.8928,E2 182.6244} C_DIS
LIN {X -11.3951,Y -132.3078,Z 175,A -92.4874,B 7.8928,C 0.3819,E1 7.8887,E2 184.0979} C_DIS
LIN {X -14.6337,Y -131.9893,Z 175,A -93.8908,B 7.8928,C 0.3816,E1 7.8848,E2 185.5018} C_DIS
LIN {X -17.8821,Y -131.5894,Z 175,A -95.3013,B 7.8928,C 0.3813,E1 7.8809,E2 186.9127} C_DIS
LIN {X -21.1024,Y -131.1121,Z 175,A -96.7021,B 7.8928,C 0.3807,E1 7.8771,E2 188.3135} C_DIS
LIN {X -23.997,Y -130.6125,Z 175,A -97.9502,B 7.8928,C 0.3799,E1 7.8736,E2 189.5596} C_DIS
LIN {X -27.1876,Y -129.9864,Z 175,A -99.3911,B 7.8928,C 0.3799,E1 7.8697,E2 191.0055} C_DIS
LIN {X -29.779,Y -129.4154,Z 175,A -100.597,B 7.8928,C 0.3803,E1 7.8664,E2 192.2191} C_DIS
LIN {X -33.3141,Y -128.5523,Z 175,A -102.2005,B 7.8928,C 0.3799,E1 7.862,E2 193.8272} C_DIS
LIN {X -36.7616,Y -127.6088,Z 175,A -103.6681,B 7.893,C 0.3777,E1 7.8581,E2 195.286} C_DIS
LIN {X -39.8429,Y -126.6806,Z 175,A -105.2175,B 7.893,C 0.3792,E1 7.8539,E2 196.8553} C_DIS
LIN {X -44.1164,Y -125.2567,Z 175,A -107.024,B 7.893,C 0.3755,E1 7.8492,E2 198.6454} C_DIS
LIN {X -47.5038,Y -124.0116,Z 175,A -108.6792,B 7.893,C 0.3756,E1 7.8448,E2 200.3128} C_DIS
LIN {X -50.8194,Y -122.689,Z 175,A -110.019,B 7.8933,C 0.371,E1 7.8414,E2 201.6282} C_DIS
LIN {X -53.5287,Y -121.5331,Z 175,A -111.4117,B 7.8933,C 0.3716,E1 7.8378,E2 203.036} C_DIS
LIN {X -56.7765,Y -120.0489,Z 175,A -112.965,B 7.8933,C 0.3701,E1 7.8339,E2 204.5909} C_DIS
LIN {X -59.4201,Y -118.7638,Z 175,A -114.2559,B 7.8934,C 0.3689,E1 7.8306,E2 205.8846} C_DIS
LIN {X -62.3133,Y -117.2711,Z 175,A -115.5497,B 7.8936,C 0.3655,E1 7.8274,E2 207.1649} C_DIS
LIN {X -65.4651,Y -115.5424,Z 175,A -117.227,B 7.8936,C 0.3655,E1 7.8233,E2 208.8577} C_DIS
LIN {X -68.277,Y -113.9032,Z 175,A -118.6497,B 7.8936,C 0.3638,E1 7.8199,E2 210.2825} C_DIS
LIN {X -71.0483,Y -112.1951,Z 175,A -120.0017,B 7.8938,C 0.361,E1 7.8167,E2 211.628} C_DIS
LIN {X -73.777,Y -110.4197,Z 175,A -121.4026,B 7.8938,C 0.3588,E1 7.8134,E2 213.0284} C_DIS
LIN {X -76.4858,Y -108.561,Z 175,A -122.9093,B 7.8939,C 0.3579,E1 7.8099,E2 214.5457} C_DIS
LIN {X -79.1157,Y -106.6599,Z 175,A -124.3207,B 7.8939,C 0.3559,E1 7.8068,E2 215.9583} C_DIS
LIN {X -81.6988,Y -104.695,Z 175,A -125.7837,B 7.8941,C 0.3544,E1 7.8035,E2 217.4288} C_DIS
LIN {X -84.756,Y -102.235,Z 175,A -127.485,B 7.8941,C 0.3516,E1 7.7998,E2 219.1306} C_DIS
LIN {X -87.8489,Y -99.5899,Z 175,A -129.27,B 7.8943,C 0.3489,E1 7.7961,E2 220.9188} C_DIS
LIN {X -90.8699,Y -96.8419,Z 175,A -131.0497,B 7.8944,C 0.3458,E1 7.7924,E2 222.7003} C_DIS
LIN {X -93.7926,Y -94.0137,Z 175,A -132.8499,B 7.8946,C 0.3431,E1 7.7888,E2 224.5055} C_DIS
LIN {X -96.7496,Y -90.9677,Z 175,A -134.7839,B 7.8946,C 0.3409,E1 7.785,E2 226.4512} C_DIS
LIN {X -99.8504,Y -87.5532,Z 175,A -136.7589,B 7.8948,C 0.3365,E1 7.7814,E2 228.4237} C_DIS
LIN {X -102.672,Y -84.2263,Z 175,A -138.6992,B 7.895,C 0.3333,E1 7.7779,E2 230.3704} C_DIS
LIN {X -105.1998,Y -81.0476,Z 175,A -140.4632,B 7.8951,C 0.3296,E1 7.7749,E2 232.1351} C_DIS
LIN {X -107.4431,Y -78.0484,Z 175,A -141.9282,B 7.8954,C 0.3238,E1 7.7725,E2 233.5811} C_DIS
LIN {X -109.3203,Y -75.3972,Z 175,A -143.4871,B 7.8954,C 0.3228,E1 7.7699,E2 235.1584} C_DIS
LIN {X -111.6473,Y -71.9067,Z 175,A -145.3973,B 7.8955,C 0.3199,E1 7.767,E2 237.0798} C_DIS
LIN {X -113.739,Y -68.5496,Z 175,A -147.0005,B 7.8957,C 0.3144,E1 7.7647,E2 238.6697} C_DIS
LIN {X -115.4099,Y -65.6972,Z 175,A -148.437,B 7.8959,C 0.311,E1 7.7627,E2 240.1067} C_DIS
LIN {X -117.1255,Y -62.5881,Z 175,A -150.0164,B 7.896,C 0.3078,E1 7.7605,E2 241.6909} C_DIS
LIN {X -118.6184,Y -59.7081,Z 175,A -151.4239,B 7.8961,C 0.3044,E1 7.7588,E2 243.0986} C_DIS
LIN {X -119.9051,Y -57.0775,Z 175,A -152.7486,B 7.8962,C 0.302,E1 7.7571,E2 244.4299} C_DIS
LIN {X -121.4045,Y -53.8162,Z 175,A -154.3066,B 7.8964,C 0.2981,E1 7.7553,E2 245.988} C_DIS
LIN {X -123.0753,Y -49.8755,Z 175,A -156.2203,B 7.8965,C 0.2942,E1 7.7533,E2 247.9086} C_DIS
LIN {X -124.4791,Y -46.2614,Z 175,A -157.8506,B 7.8967,C 0.2892,E1 7.7517,E2 249.5327} C_DIS
LIN {X -125.5753,Y -43.1974,Z 175,A -159.241,B 7.8968,C 0.2852,E1 7.7504,E2 250.9206} C_DIS
LIN {X -126.5961,Y -40.1072,Z 175,A -160.7171,B 7.8969,C 0.2823,E1 7.7491,E2 252.4042} C_DIS
LIN {X -127.5876,Y -36.8337,Z 175,A -162.2143,B 7.8971,C 0.2786,E1 7.7479,E2 253.9031} C_DIS
LIN {X -128.4301,Y -33.7786,Z 175,A -163.6075,B 7.8972,C 0.2752,E1 7.7469,E2 255.2983} C_DIS
LIN {X -129.2097,Y -30.662,Z 175,A -164.9878,B 7.8973,C 0.2712,E1 7.746,E2 256.6769} C_DIS
LIN {X -130.1053,Y -26.6035,Z 175,A -166.9196,B 7.8974,C 0.2681,E1 7.7448,E2 258.6239} C_DIS
LIN {X -130.8436,Y -22.7058,Z 175,A -168.5828,B 7.8976,C 0.2626,E1 7.744,E2 260.28} C_DIS
LIN {X -131.3135,Y -19.8028,Z 175,A -169.8762,B 7.8977,C 0.2593,E1 7.7435,E2 261.5754} C_DIS
LIN {X -131.7603,Y -16.578,Z 175,A -171.3093,B 7.8979,C 0.2557,E1 7.7429,E2 263.0108} C_DIS
LIN {X -132.1278,Y -13.3348,Z 175,A -172.7707,B 7.8979,C 0.2524,E1 7.7425,E2 264.4774} C_DIS
LIN {X -132.4143,Y -10.0888,Z 175,A -174.267,B 7.898,C 0.2495,E1 7.7422,E2 265.9832} C_DIS
LIN {X -132.6214,Y -6.8391,Z 175,A -175.6758,B 7.8982,C 0.2455,E1 7.7419,E2 267.3913} C_DIS
LIN {X -132.7539,Y -3.4147,Z 175,A -177.1271,B 7.8983,C 0.2409,E1 7.7419,E2 268.8381} C_DIS
LIN {X -132.7991,Y -0.2336,Z 175,A -178.5839,B 7.8983,C 0.2381,E1 7.7418,E2 270.3037} C_DIS
LIN {X -132.767,Y 2.9407,Z 175,A -179.94,B 7.8985,C 0.234,E1 7.7418,E2 271.6571} C_DIS
LIN {X -132.6538,Y 6.1948,Z 175,A 178.5628,B 7.8986,C 0.2311,E1 7.742,E2 273.1639} C_DIS
LIN {X -132.4613,Y 9.4453,Z 175,A 177.245,B 7.8988,C 0.2259,E1 7.7422,E2 274.4701} C_DIS
LIN {X -132.1583,Y 13.0171,Z 175,A 175.649,B 7.8988,C 0.2221,E1 7.7426,E2 276.0705} C_DIS
LIN {X -131.7999,Y 16.2542,Z 175,A 174.2203,B 7.899,C 0.2184,E1 7.7431,E2 277.5008} C_DIS
LIN {X -131.3623,Y 19.4829,Z 175,A 172.7885,B 7.899,C 0.2147,E1 7.7437,E2 278.9344} C_DIS
LIN {X -130.8983,Y 22.3839,Z 175,A 171.493,B 7.8992,C 0.2115,E1 7.7443,E2 280.2319} C_DIS
LIN {X -130.2485,Y 25.8994,Z 175,A 169.9996,B 7.8992,C 0.2065,E1 7.745,E2 281.7181} C_DIS
LIN {X -129.6359,Y 28.8138,Z 175,A 168.5009,B 7.8993,C 0.2057,E1 7.7459,E2 283.2409} C_DIS
LIN {X -128.8915,Y 31.9778,Z 175,A 167.1711,B 7.8994,C 0.2008,E1 7.7468,E2 284.5607} C_DIS
LIN {X -128.07,Y 35.1228,Z 175,A 165.7442,B 7.8995,C 0.1972,E1 7.7478,E2 285.9892} C_DIS
LIN {X -127.1715,Y 38.2479,Z 175,A 164.385,B 7.8996,C 0.1927,E1 7.7489,E2 287.3419} C_DIS
LIN {X -126.1967,Y 41.3506,Z 175,A 162.7955,B 7.8996,C 0.1913,E1 7.7503,E2 288.9521} C_DIS
LIN {X -125.1464,Y 44.4282,Z 175,A 161.4625,B 7.8998,C 0.1865,E1 7.7515,E2 290.2754} C_DIS
LIN {X -124.0215,Y 47.4782,Z 175,A 159.9318,B 7.8998,C 0.1844,E1 7.753,E2 291.8198} C_DIS
LIN {X -122.6898,Y 50.8175,Z 175,A 158.5734,B 7.9,C 0.1777,E1 7.7544,E2 293.154} C_DIS
LIN {X -121.5284,Y 53.5391,Z 175,A 157.1809,B 7.9,C 0.1758,E1 7.756,E2 294.5589} C_DIS
LIN {X -120.0449,Y 56.7848,Z 175,A 155.5934,B 7.9,C 0.1724,E1 7.7578,E2 296.1505} C_DIS
LIN {X -118.7602,Y 59.4274,Z 175,A 154.2898,B 7.9002,C 0.1696,E1 7.7594,E2 297.4572} C_DIS
LIN {X -117.4267,Y 62.0168,Z 175,A 152.9775,B 7.9002,C 0.1671,E1 7.7612,E2 298.7747} C_DIS
LIN {X -115.5063,Y 65.5283,Z 175,A 151.2758,B 7.9003,C 0.1624,E1 7.7635,E2 300.4719} C_DIS
LIN {X -113.8853,Y 68.3069,Z 175,A 149.8499,B 7.9003,C 0.1594,E1 7.7655,E2 301.9008} C_DIS
LIN {X -112.1906,Y 71.0554,Z 175,A 148.5009,B 7.9004,C 0.1554,E1 7.7675,E2 303.2433} C_DIS
LIN {X -110.4269,Y 73.7662,Z 175,A 147.1064,B 7.9005,C 0.152,E1 7.7696,E2 304.6363} C_DIS
LIN {X -108.6007,Y 76.4295,Z 175,A 145.5965,B 7.9005,C 0.1503,E1 7.772,E2 306.1586} C_DIS
LIN {X -106.6669,Y 79.1063,Z 175,A 144.0048,B 7.9005,C 0.1492,E1 7.7747,E2 307.7685} C_DIS
LIN {X -104.0895,Y 82.4684,Z 175,A 142.1703,B 7.9006,C 0.1451,E1 7.7778,E2 309.602} C_DIS
LIN {X -101.1856,Y 86.006,Z 175,A 140.2998,B 7.9007,C 0.1393,E1 7.7812,E2 311.4583} C_DIS
LIN {X -98.8383,Y 88.6937,Z 175,A 138.6097,B 7.9007,C 0.138,E1 7.7843,E2 313.1647} C_DIS
LIN {X -96.1783,Y 91.5716,Z 175,A 136.8966,B 7.9008,C 0.1348,E1 7.7876,E2 314.8788} C_DIS
LIN {X -93.3173,Y 94.4859,Z 175,A 135.0959,B 7.9008,C 0.1317,E1 7.7911,E2 316.6824} C_DIS
LIN {X -90.3831,Y 97.2958,Z 175,A 133.3318,B 7.9009,C 0.1283,E1 7.7947,E2 318.4462} C_DIS
LIN {X -87.364,Y 100.0155,Z 175,A 131.6503,B 7.9009,C 0.124,E1 7.7982,E2 320.1177} C_DIS
LIN {X -84.2393,Y 102.6615,Z 175,A 129.7702,B 7.901,C 0.1223,E1 7.8023,E2 322.0094} C_DIS
Enddeposition()
END
